(* Call ST03_572_Y70_0  Zuführung Vereinzler AST/GST  (Valve) *)
Analyze(InputExp:=  TRUE, DoAnalyze:= TRUE );
ST03_572_Y70_0.strAnlayse:=Analyze.OutString;
ST03_572_Y70_0(Enable  :=  Analyze.ExpResult,
                                sVisu:=Visu.ST03_572_Y70_0,
                                Reset:=gResetAll,
);
ST03_571_B69_2(ValveObject:= ADR(ST03_572_Y70_0));(*  Zuführung Vereinzler eingefahren GST*)
ST03_571_B69_3(ValveObject:= ADR(ST03_572_Y70_0));(*  Zuführung Vereinzler ausgefahren AST*)

(* Call ST03_572_Y70_1  Züführung Stopper AST/GST  (Valve) *)
Analyze(InputExp:=  TRUE, DoAnalyze:= TRUE );
ST03_572_Y70_1.strAnlayse:=Analyze.OutString;
ST03_572_Y70_1(Enable  :=  Analyze.ExpResult,
                                sVisu:=Visu.ST03_572_Y70_1,
                                Reset:=gResetAll,
);
ST03_571_B69_4(ValveObject:= ADR(ST03_572_Y70_1));(* Zuführung Stopper  eingefahren  AST*)
ST03_571_B69_5(ValveObject:= ADR(ST03_572_Y70_1));(* Zuführung Stopper  ausgefahren GST*)


(* Call ST03_571_B69_6 SK anwesend am Stoper (DigIn) *)
ST03_571_B69_6(sVisu:=Visu.ST03_571_B69_6,
                                Reset:=gResetAll,
);
(* Call ST03_571_B69_7 ISK anwesend an Abholposition (DigIn) *)
ST03_571_B69_7(sVisu:=Visu.ST03_571_B69_7,
                                Reset:=gResetAll,
);
END_ACTION
ACTION call_46pol:
(* Call ST03_463_Y71_3 Förderband  Zuführung Vereinzler AST/GST  (Valve) *)
Analyze(InputExp:=  TRUE, DoAnalyze:= TRUE );
ST03_464_Y71_3.strAnlayse:=Analyze.OutString;
ST03_464_Y71_3(Enable  :=  Analyze.ExpResult,
                                sVisu:=Visu.ST03_464_Y71_3,
                                Reset:=gResetAll,
);
ST03_461_B69_0(ValveObject:= ADR(ST03_464_Y71_3));(*Förderband Zuführung Vereinzler   AST*)
ST03_461_B69_1(ValveObject:= ADR(ST03_464_Y71_3));(*Förderband Zuführung Vereinzler   GST*)

(* Call ST03_463_Y71_4 Förderband  Zuführung Stopper AST/GST  (Valve) *)
Analyze(InputExp:=  TRUE, DoAnalyze:= TRUE );
ST03_464_Y71_4.strAnlayse:=Analyze.OutString;
ST03_464_Y71_4(Enable  :=  Analyze.ExpResult,
                                sVisu:=Visu.ST03_464_Y71_4,
                                Reset:=gResetAll,
);
ST03_461_B69_2(ValveObject:= ADR(ST03_464_Y71_4));(*Förderband Zuführung Stopper   AST*)
ST03_461_B69_3(ValveObject:= ADR(ST03_464_Y71_4));(*Förderband Zuführung Stopper   GST*)

(* Call ST03_461_B69_4 Zuführung  frei zum Ablegen ISK SP Maschine Pos.1  (DigIn) *)
ST03_461_B69_4(sVisu:=Visu.ST03_461_B69_4,
                                Reset:=gResetAll,
);
(* Call ST03_461_B69_7 Zuführung  ISK anwesend am Stopper (DigIn) *)
ST03_461_B69_7(sVisu:=Visu.ST03_461_B69_7,
                                Reset:=gResetAll,
);
(* Call ST03_463_B70_7  ISK auf Übergabeposition zu Roboter  (DigIn) *)
ST03_463_B70_7(sVisu:=Visu.ST03_463_B70_7,
                                Reset:=gResetAll,
);
(* Call ST03_462_B70_0 Förderband  ISK anwesend Wender (DigIn) *)
ST03_462_B70_0(sVisu:=Visu.ST03_462_B70_0,
                                Reset:=gResetAll,
);
(* Call ST03_462_B70_1 Zuführung  ISK Lageerkennung rechts (DigIn) *)
ST03_462_B70_1(sVisu:=Visu.ST03_462_B70_1,
                                Reset:=gResetAll,
);
(* Call ST03_462_B70_2 Zuführung  ISK Lageerkennung links (DigIn) *)
ST03_462_B70_2(sVisu:=Visu.ST03_462_B70_2,
                                Reset:=gResetAll,
);
(* Call ST03_464_Y71_0 Förderband  Zuführung Vereinzelner Wender AST/GST  (Valve) *)
Analyze(InputExp:=  TRUE, DoAnalyze:= TRUE );
ST03_464_Y71_0.strAnlayse:=Analyze.OutString;
ST03_464_Y71_0(Enable  :=  Analyze.ExpResult,
                                sVisu:=Visu.ST03_464_Y71_0,
                                Reset:=gResetAll,
);
ST03_461_B69_5(ValveObject:= ADR(ST03_464_Y71_0));(*Förderbandeinheit  Zuführung  Vereinzelner Wender AST*)
ST03_461_B69_6(ValveObject:= ADR(ST03_464_Y71_0));(*Förderbandeinheit  Zuführung  Vereinzelner Wender GST*)

(* Call ST03_464_Y71_1 Förderband  Zuführung Zylinder Vakuumdüsen AST/GST  (Valve) *)
Analyze(InputExp:=  TRUE, DoAnalyze:= TRUE );
ST03_464_Y71_1.strAnlayse:=Analyze.OutString;
ST03_464_Y71_1(Enable  :=  Analyze.ExpResult,
                                sVisu:=Visu.ST03_464_Y71_1,
                                Reset:=gResetAll,
);
ST03_463_B70_3(ValveObject:= ADR(ST03_464_Y71_1));(*Förderband Zuführung Zylinder Vakuumdüsen   AST*)
ST03_463_B70_4(ValveObject:= ADR(ST03_464_Y71_1));(*Förderband Zuführung Zylinder Vakuumdüsen   GST*)

IF	ST03_463_B70_3.ValveSensor THEN
	ST03_463_B70_3_4_pos:= -14;
ELSIF
	ST03_463_B70_4.ValveSensor THEN
	ST03_463_B70_3_4_pos:= 0;
ELSE
	ST03_463_B70_3_4_pos:= -7;
END_IF

(* Call ST03_464_Y71_2  Förderband  Zuführung Wendestation Einlauf / Auslauf   (Valve) *)
Analyze(InputExp:=  TRUE, DoAnalyze:= TRUE );
ST03_464_Y71_2.strAnlayse:=Analyze.OutString;
ST03_464_Y71_2(Enable  :=  Analyze.ExpResult,
                                sVisu:=Visu.ST03_464_Y71_2,
                                Reset:=gResetAll,
);
ST03_463_B70_5(ValveObject:= ADR(ST03_464_Y71_2));(*Förderband Zuführung Wendestation   AST*)
ST03_463_B70_6(ValveObject:= ADR(ST03_464_Y71_2));(*Förderband Zuführung Wendestation   GST*)

(* Call ST03_464_Y71_5  Förderband  Zuführung Vakuumdüsen EIN/AUS  (Valve) *)
Analyze(InputExp:=  TRUE, DoAnalyze:= TRUE );
ST03_464_Y71_5.strAnlayse:=Analyze.OutString;
ST03_464_Y71_5(Enable  :=  Analyze.ExpResult,
                                sVisu:=Visu.ST03_464_Y71_5,
                                Reset:=gResetAll,
);
(* Call ST03_464_B71_6  Vakuum vorhanden (DigIn) *)
ST03_464_B71_6(sVisu:=Visu.ST03_464_B71_6,
                                Reset:=gResetAll,
);
(* Call ST03_464_B71_7 Förderband  Staustrecke mitte voll (DigIn) *)
ST03_464_B71_7(sVisu:=Visu.ST03_464_B71_7,
                                Reset:=gResetAll,
);
END_ACTION
ACTION call_48pol:
(* Call ST03_551_B69_0 IZuführung  frei zum Ablegen ISK SP Maschine (DigIn) *)
ST03_551_B69_0(sVisu:=Visu.ST03_551_B69_0,
                                Reset:=gResetAll,
);
(* Call ST03_552_Y70_1  Zuführung Vereinzler AST/GST  (Valve) *)
Analyze(InputExp:=  TRUE, DoAnalyze:= TRUE );
ST03_552_Y70_1.strAnlayse:=Analyze.OutString;
ST03_552_Y70_1(Enable  :=  Analyze.ExpResult,
                                sVisu:=Visu.ST03_552_Y70_1,
                                Reset:=gResetAll,
);
ST03_551_B69_1(ValveObject:= ADR(ST03_552_Y70_1));(*  Zuführung Vereinzler eingefahren GST*)
ST03_551_B69_2(ValveObject:= ADR(ST03_552_Y70_1));(*  Zuführung Vereinzler ausgefahren AST*)

(* Call ST03_552_Y70_2  Züführung Stopper AST/GST  (Valve) *)
Analyze(InputExp:=  TRUE, DoAnalyze:= TRUE );
ST03_552_Y70_2.strAnlayse:=Analyze.OutString;
ST03_552_Y70_2(Enable  :=  Analyze.ExpResult,
                                sVisu:=Visu.ST03_552_Y70_2,
                                Reset:=gResetAll,
);
ST03_551_B69_3(ValveObject:= ADR(ST03_552_Y70_2));(* Zuführung Stopper  eingefahren  AST*)
ST03_551_B69_4(ValveObject:= ADR(ST03_552_Y70_2));(* Zuführung Stopper  ausgefahren GST*)


(* Call ST03_551_B69_6 SK anwesend am Stoper (DigIn) *)
ST03_551_B69_6(sVisu:=Visu.ST03_551_B69_6,
                                Reset:=gResetAll,
);
(* Call ST03_541_B69_7 ISK Lageerkennung links (DigIn) *)
ST03_551_B69_7(sVisu:=Visu.ST03_551_B69_7,
                                Reset:=gResetAll,
);
(* Call ST03_542_B70_0  ISK Lageerkennung rechts (DigIn) *)
ST03_552_B70_0(sVisu:=Visu.ST03_552_B70_0,
                                Reset:=gResetAll,
);
END_ACTION
ACTION call_72pol:
(* Call ST03_546_B69_0 IZuführung  frei zum Ablegen ISK SP Maschine (DigIn) *)
ST03_546_B69_0(sVisu:=Visu.ST03_546_B69_0,
                                Reset:=gResetAll,
);
(* Call ST03_547_Y70_1  Zuführung Vereinzler AST/GST  (Valve) *)
Analyze(InputExp:=  TRUE, DoAnalyze:= TRUE );
ST03_547_Y70_1.strAnlayse:=Analyze.OutString;
ST03_547_Y70_1(Enable  :=  Analyze.ExpResult,
                                sVisu:=Visu.ST03_547_Y70_1,
                                Reset:=gResetAll,
);
ST03_546_B69_1(ValveObject:= ADR(ST03_547_Y70_1));(*  Zuführung Vereinzler eingefahren GST*)
ST03_546_B69_2(ValveObject:= ADR(ST03_547_Y70_1));(*  Zuführung Vereinzler ausgefahren AST*)

(* Call ST03_547_Y70_2  Züführung Stopper AST/GST  (Valve) *)
Analyze(InputExp:=  TRUE, DoAnalyze:= TRUE );
ST03_547_Y70_2.strAnlayse:=Analyze.OutString;
ST03_547_Y70_2(Enable  :=  Analyze.ExpResult,
                                sVisu:=Visu.ST03_547_Y70_2,
                                Reset:=gResetAll,
);
ST03_546_B69_3(ValveObject:= ADR(ST03_547_Y70_2));(* Zuführung Stopper  eingefahren  AST*)
ST03_546_B69_4(ValveObject:= ADR(ST03_547_Y70_2));(* Zuführung Stopper  ausgefahren GST*)


(* Call ST03_546_B69_6 SK anwesend am Stoper (DigIn) *)
ST03_546_B69_6(sVisu:=Visu.ST03_546_B69_6,
                                Reset:=gResetAll,
);
(* Call ST03_546_B69_7 ISK anwesend an Abholposition (DigIn) *)
ST03_546_B69_7(sVisu:=Visu.ST03_546_B69_7,
                                Reset:=gResetAll,
);
(* Call ST03_547_B70_0  ISK Lageerkennung (DigIn) *)
ST03_547_B70_0(sVisu:=Visu.ST03_547_B70_0,
                                Reset:=gResetAll,
);
END_ACTION
ACTION call_74_91_35_168_160pol:
(* Call ST03_421_B63_4 Förderband frei zum Ablegen ISK SP Maschine Pos1  (DigIn) *)
ST03_421_B63_4(sVisu:=Visu.ST03_421_B63_4,
                                Reset:=gResetAll,
);
(* Call ST03_421_B63_5 Förderband frei zum Ablegen ISK SP Maschine Pos2  (DigIn) *)
ST03_421_B63_5(sVisu:=Visu.ST03_421_B63_5,
                                Reset:=gResetAll,
);
(* Call ST03_421_B63_6 Förderband frei zum Ablegen ISK SP Maschine Pos3  (DigIn) *)
ST03_421_B63_6(sVisu:=Visu.ST03_421_B63_6,
                                Reset:=gResetAll,
);
(* Call ST03_421_B63_7 ISK anwesend am Vereinzler  (DigIn) *)
ST03_421_B63_7(sVisu:=Visu.ST03_421_B63_7,
                                Reset:=gResetAll,
);
(* Call ST03_422_B64_0 Förderband Trigger Tintenstrahldrucker (Lichtschranke)  (DigIn) *)
ST03_422_B64_0(sVisu:=Visu.ST03_422_B64_0,
                                Reset:=gResetAll,
);
(* Call ST03_423_B66_0 Förderband Trigger Tintenstrahldrucker (Lichtschranke)  (DigIn) *)
ST03_423_B66_0(sVisu:=Visu.ST03_423_B66_0,
                                Reset:=gResetAll,
);
(* Call ST03_8_B76_1 Förderband Trigger Tintenstrahldrucker (Lichtschranke)  (DigIn) 3621 *)
ST03_8_B76_1(sVisu:=Visu.ST03_8_B76_1,
                                Reset:=gResetAll,
);
(* Call ST03_8_B76_2 Förderband Trigger Tintenstrahldrucker (Lichtschranke)  (DigIn) 3621 *)
ST03_8_B76_2(sVisu:=Visu.ST03_8_B76_2,
                                Reset:=gResetAll,
);
(* Call ST03_422_B64_3  Förderband ISK anwesend Stopper Kamera  (DigIn) *)
ST03_422_B64_3(sVisu:=Visu.ST03_422_B64_3,
                                Reset:=gResetAll,
);
(* Call ST03_422_B64_4 Zuführung ISK auf Übergabeposition Robo Palettierer  (DigIn) *)
ST03_422_B64_4(sVisu:=Visu.ST03_422_B64_4,
                                Reset:=gResetAll,
);
(* Call ST03_422_Y64_5  Förderband  Zuführung Vereinzler AST/GST (Valve) *)
Analyze(InputExp:=  TRUE, DoAnalyze:= TRUE );
ST03_422_Y64_5.strAnlayse:=Analyze.OutString;
ST03_422_Y64_5(Enable  :=  Analyze.ExpResult,
                                sVisu:=Visu.ST03_422_Y64_5,
                                Reset:=gResetAll,
);
ST03_421_B63_0(ValveObject:= ADR(ST03_422_Y64_5));(*Förderband Zuführung Vereinzler AST*)
ST03_421_B63_1(ValveObject:= ADR(ST03_422_Y64_5));(*Förderband Zuführung Vereinzler GST*)

(* Call ST03_422_Y64_6 Förderband rechte Zuführung Vereinzler AST/GST (Valve) *)
Analyze(InputExp:=  TRUE, DoAnalyze:= TRUE );
ST03_422_Y64_6.strAnlayse:=Analyze.OutString;
ST03_422_Y64_6(Enable  :=  Analyze.ExpResult,
                                sVisu:=Visu.ST03_422_Y64_6,
                                Reset:=gResetAll,
);
ST03_421_B63_2(ValveObject:= ADR(ST03_422_Y64_6));(*Förderband Zuführung Stopper AST*)
ST03_421_B63_3(ValveObject:= ADR(ST03_422_Y64_6));(*Förderband Zuführung Stopper GST*)

(* Call ST03_422_Y64_7 Förderband links/rechts Züführung Stopper 1 AST/GST (Valve) *)
Analyze(InputExp:=  TRUE, DoAnalyze:= TRUE );
ST03_422_Y64_7.strAnlayse:=Analyze.OutString;
ST03_422_Y64_7(Enable  :=  Analyze.ExpResult,
                                sVisu:=Visu.ST03_422_Y64_7,
                                Reset:=gResetAll,
);
ST03_422_B64_2(ValveObject:= ADR(ST03_422_Y64_7));(*Förderband Zuführung Stopper Kamera AST*)
ST03_422_B64_1(ValveObject:= ADR(ST03_422_Y64_7));(*Förderband Zuführung Stopper Kamera GST*)


(* Call ST03_423_Y65_6 Förderband links/rechts Züführung Stopper 2 AST/GST (Valve) *)
Analyze(InputExp:=  TRUE, DoAnalyze:= TRUE );
ST03_423_Y65_6.strAnlayse:=Analyze.OutString;
ST03_423_Y65_6(Enable  :=  Analyze.ExpResult,
                                sVisu:=Visu.ST03_423_Y65_6,
                                Reset:=gResetAll,
);
ST03_423_B65_1(ValveObject:= ADR(ST03_423_Y65_6));(*Förderband Zuführung Stopper Kamera AST*)
ST03_423_B65_0(ValveObject:= ADR(ST03_423_Y65_6));(*Förderband Zuführung Stopper Kamera GST*)

(* Call ST03_423_Y65_7 Förderband links/rechts Züführung Stopper 3 AST/GST (Valve) *)
Analyze(InputExp:=  TRUE, DoAnalyze:= TRUE );
ST03_423_Y65_7.strAnlayse:=Analyze.OutString;
ST03_423_Y65_7(Enable  :=  Analyze.ExpResult,
                                sVisu:=Visu.ST03_423_Y65_7,
                                Reset:=gResetAll,
);
ST03_423_B65_3(ValveObject:= ADR(ST03_423_Y65_7));(*Förderband Zuführung Stopper Kamera AST*)
ST03_423_B65_4(ValveObject:= ADR(ST03_423_Y65_7));(*Förderband Zuführung Stopper Kamera GST*)

(* Call ST03_33F4 Steckdosenleise Tintenstrahldrucker  (DigIn) *)
ST03_33F4(		sVisu:=Visu.ST03_33F4,
				Reset:=gResetAll,
);
(* Call ST03_70U3_1 Bereit/ Im Druck Tintenstrahldrucker Frontseite   (DigIn) *)
ST03_70U3_1(sVisu:=Visu.ST03_70U3_1,
                                Reset:=gResetAll,
);
(* Call ST03_70U3_2 Tank voll Tintenstrahldrucker Frontseite   (DigIn) *)
ST03_70U3_2(	sVisu:=Visu.ST03_70U3_2,
				Reset:=gResetAll,
);
(* Call ST03_70U3_3 Fehler/Störung Tintenstrahldrucker Frontseite   (DigIn) *)
ST03_70U3_3(	sVisu:=Visu.ST03_70U3_3,
				Reset:=gResetAll,
);
(* Call ST03_71U3_1 Bereit/ Im Druck Tintenstrahldrucker Rückseite   (DigIn) *)
ST03_71U3_1(sVisu:=Visu.ST03_71U3_1,
                                Reset:=gResetAll,
);
(* Call ST03_71U3_2 Tank voll Tintenstrahldrucker Rückseite   (DigIn) *)
ST03_71U3_2(	sVisu:=Visu.ST03_71U3_2,
				Reset:=gResetAll,
);
(* Call ST03_71U3_3 Fehler/Störung Tintenstrahldrucker Rückseite   (DigIn) *)
ST03_71U3_3(	sVisu:=Visu.ST03_71U3_3,
				Reset:=gResetAll,
);
(* Call ST03_PLAN_70V1_1 Start  Bedrucken Tintenstrahldrucker Frontseite (DigOutIn) *)
ST03_PLAN_70V1_1(	sVisu:=Visu.ST03_PLAN_70V1_1,
						Reset:=gResetAll,
);
(* Call ST03_PLAN_70V1_1 Start  Bedrucken Tintenstrahldrucker Rückseite (DigOutIn) *)
ST03_PLAN_71V1_2(	sVisu:=Visu.ST03_PLAN_71V1_2,
						Reset:=gResetAll,
);
IF NOT MP.ST02.SensopartEthernet THEN
	(**Sensopart Kamera links*)
	ST03_8_80_A1(
		b_kamera_aktiv:=MP.ST03.FrontCamOn,
		st_Description:= 'Sensopart Kamera links',
		b_reset:=gResetAll );

	(**Sensopart Kamera rechts*)
	ST03_8_85_A1(
		b_kamera_aktiv:=MP.ST03.BackCamOn,
		st_Description:= 'Sensopart Kamera rechts',
		b_reset:=gResetAll );
ELSE
	(**Sensopart Kamera links*)
	IF MP.ST02.SensopartIPAdress <>''  THEN
		ST03_8_90_A1(
				Activated := MP.ST03.FrontCamOn,
				st_Description:= 'Sensopart Kamera links',
				);
		ST03_8_90_A1.s_IpAdress := MP.ST02.SensopartIPAdress;
		ST03_8_90_A1.i_CmdPort := 2006;
		ST03_8_90_A1.i_DataPort :=2005;
END_IF
	(**Sensopart Kamera rechts*)
	IF MP.ST02.SensopartIPAdress2 <>''  THEN
		ST03_8_95_A1(
				Activated := MP.ST03.BackCamOn,
				st_Description:= 'Sensopart Kamera rechts',
				);
		ST03_8_95_A1.s_IpAdress := MP.ST02.SensopartIPAdress2;
		ST03_8_95_A1.i_CmdPort := 2006;
		ST03_8_95_A1.i_DataPort :=2005;
	END_IF
END_IF

(* Init ST03_S18 ST02 Druckschalter Wartungseinheit Hauptluft Tintenstrahldrucker min.6 bar (DigIn)
nur bei 160 pol*)	
ST03_S18(	sVisu:=Visu.ST03_S18,
			Reset:=gResetAll,
);
(* Call ST03_H6 Signalsäule GR Bedruckung IO(DigOutIn) *)
ST03_H6(	sVisu:=Visu.ST03_H6,
			Reset:=gResetAll,
);
(* Call ST03_H7 Signalsäule RD Sammelstörung Bedruckung IO(DigOutIn) *)
ST03_H7(	sVisu:=Visu.ST03_H7,
			Reset:=gResetAll,
);
END_ACTION
ACTION call_7pol:
(* Call ST03_512_XG1 Zuführung  frei zum Ablegen ISK SP Maschine (DigIn) *)
ST03_512_XG1(sVisu:=Visu.ST03_512_XG1,
                                Reset:=gResetAll,
);
(* Call ST03_515_Y72_0 ISK Klemmer 1 AST/GST  (Valve) *)
Analyze(InputExp:=  TRUE, DoAnalyze:= TRUE );
ST03_515_Y72_0.strAnlayse:=Analyze.OutString;
ST03_515_Y72_0(Enable  :=  Analyze.ExpResult,
                                sVisu:=Visu.ST03_515_Y72_0,
                                Reset:=gResetAll,
);
ST03_512_B69_1(ValveObject:= ADR(ST03_515_Y72_0));(*ISK Klemmer 2 GST*)
ST03_512_B69_2(ValveObject:= ADR(ST03_515_Y72_0));(*ISK Klemmer 2 AST*)
ST03_512_B69_3(ValveObject:= ADR(ST03_515_Y72_0));(*ISK Klemmer 1 GST*)
ST03_512_B69_4(ValveObject:= ADR(ST03_515_Y72_0));(*ISK Klemmer 1 AST*)

(* Call ST03_515_Y72_1 Rinne schwenkern AST/GST  (Valve) *)
Analyze(InputExp:=  TRUE, DoAnalyze:= TRUE );
ST03_515_Y72_1.strAnlayse:=Analyze.OutString;
ST03_515_Y72_1(Enable  :=  Analyze.ExpResult,
                                sVisu:=Visu.ST03_515_Y72_1,
                                Reset:=gResetAll,
);
ST03_512_B69_5(ValveObject:= ADR(ST03_515_Y72_1));(*ISK Klemmer schwenkern 0° AST*)
ST03_512_B69_6(ValveObject:= ADR(ST03_515_Y72_1));(*ISK Klemmer schwenkern 180° GST*)

(* Call ST03_514_B71_7 Führungsschiene frei zum schwenken (DigIn) *)
ST03_514_B71_7(sVisu:=Visu.ST03_514_B71_7,
                                Reset:=gResetAll,
);
(* Call ST03_515_Y72_2 Führungsschiene  Zuführung Vereinzler AST/GST  (Valve) *)
Analyze(InputExp:=  TRUE, DoAnalyze:= TRUE );
ST03_515_Y72_2.strAnlayse:=Analyze.OutString;
ST03_515_Y72_2(Enable  :=  Analyze.ExpResult,
                                sVisu:=Visu.ST03_515_Y72_2,
                                Reset:=gResetAll,
);
ST03_513_B70_0(ValveObject:= ADR(ST03_515_Y72_2));(*Führungsschiene  Zuführung Vereinzler AST*)
ST03_513_B70_1(ValveObject:= ADR(ST03_515_Y72_2));(*Führungsschiene  Zuführung Vereinzler GST*)

(* Call ST03_515_Y72_3 Führungsschiene  Zuführung Stopper AST/GST  (Valve) *)
Analyze(InputExp:=  TRUE, DoAnalyze:= TRUE );
ST03_515_Y72_3.strAnlayse:=Analyze.OutString;
ST03_515_Y72_3(Enable  :=  Analyze.ExpResult,
                                sVisu:=Visu.ST03_515_Y72_3,
                                Reset:=gResetAll,
);
ST03_513_B70_2(ValveObject:= ADR(ST03_515_Y72_3));(*Führungsschiene  Zuführung Stopper AST*)
ST03_513_B70_3(ValveObject:= ADR(ST03_515_Y72_3));(*Führungsschiene  Zuführung Stopper GST*)

(* Call ST03_513_B70_4 ISK anwesend am Stopper(DigIn) *)
ST03_513_B70_4(sVisu:=Visu.ST03_513_B70_4,
                                Reset:=gResetAll,
);
(* Call ST03_515_Y72_4 Übergabeposition Stopper 1 AST/GST  (Valve) *)
Analyze(InputExp:=  TRUE, DoAnalyze:= TRUE );
ST03_515_Y72_4.strAnlayse:=Analyze.OutString;
ST03_515_Y72_4(Enable  :=  Analyze.ExpResult,
                                sVisu:=Visu.ST03_515_Y72_4,
                                Reset:=gResetAll,
);
ST03_513_B70_5(ValveObject:= ADR(ST03_515_Y72_4));(*Übergabeposition Stopper 1 AST*)
ST03_513_B70_6(ValveObject:= ADR(ST03_515_Y72_4));(*Übergabeposition Stopper 1 GST*)

(* Call ST03_513_B70_7 ISK auf Übergabeposition 1 (DigIn) *)
ST03_513_B70_7(sVisu:=Visu.ST03_513_B70_7,
                                Reset:=gResetAll,
);
(* Call ST03_515_Y72_5 Übergabeposition Stopper 2 AST/GST  (Valve) *)
Analyze(InputExp:=  TRUE, DoAnalyze:= TRUE );
ST03_515_Y72_5.strAnlayse:=Analyze.OutString;
ST03_515_Y72_5(Enable  :=  Analyze.ExpResult,
                                sVisu:=Visu.ST03_515_Y72_5,
                                Reset:=gResetAll,
);
ST03_514_B71_0(ValveObject:= ADR(ST03_515_Y72_5));(*Übergabeposition Stopper 2 AST*)
ST03_514_B71_1(ValveObject:= ADR(ST03_515_Y72_5));(*Übergabeposition Stopper 2 GST*)

(* Call ST03_514_B71_2 ISK auf Übergabeposition 2 (DigIn) *)
ST03_514_B71_2(sVisu:=Visu.ST03_514_B71_2,
                                Reset:=gResetAll,
);
(* Call ST03_515_Y72_6 Übergabeposition Stopper 3 AST/GST  (Valve) *)
Analyze(InputExp:=  TRUE, DoAnalyze:= TRUE );
ST03_515_Y72_6.strAnlayse:=Analyze.OutString;
ST03_515_Y72_6(Enable  :=  Analyze.ExpResult,
                                sVisu:=Visu.ST03_515_Y72_6,
                                Reset:=gResetAll,
);
ST03_514_B71_3(ValveObject:= ADR(ST03_515_Y72_6));(*Übergabeposition Stopper 3 AST*)
ST03_514_B71_4(ValveObject:= ADR(ST03_515_Y72_6));(*Übergabeposition Stopper 3 GST*)

(* Call ST03_514_B71_5 ISK auf Übergabeposition 3 (DigIn) *)
ST03_514_B71_5(sVisu:=Visu.ST03_514_B71_5,
                                Reset:=gResetAll,
);
(* Call ST03_514_B71_6 ISK auf Übergabeposition 4 (DigIn) *)
ST03_514_B71_6(sVisu:=Visu.ST03_514_B71_6,
                                Reset:=gResetAll,
);
END_ACTION
ACTION call_88pol:
(* Call ST03_501_B69_0 IZuführung  frei zum Ablegen ISK SP Maschine (DigIn) *)
ST03_501_B69_0(sVisu:=Visu.ST03_501_B69_0,
                                Reset:=gResetAll,
);
(* Call ST03_502_Y70_1 Förderband  Zuführung Vereinzler AST/GST  (Valve) *)
Analyze(InputExp:=  TRUE, DoAnalyze:= TRUE );
ST03_502_Y70_1.strAnlayse:=Analyze.OutString;
ST03_502_Y70_1(Enable  :=  Analyze.ExpResult,
                                sVisu:=Visu.ST03_502_Y70_1,
                                Reset:=gResetAll,
);
ST03_501_B69_1(ValveObject:= ADR(ST03_502_Y70_1));(*Förderband Zuführung Vereinzler   AST*)
ST03_501_B69_2(ValveObject:= ADR(ST03_502_Y70_1));(*Förderband Zuführung Vereinzler   GST*)

(* Call ST03_502_Y70_2 örderband  Züführung Stopper AST/GST  (Valve) *)
Analyze(InputExp:=  TRUE, DoAnalyze:= TRUE );
ST03_502_Y70_2.strAnlayse:=Analyze.OutString;
ST03_502_Y70_2(Enable  :=  Analyze.ExpResult,
                                sVisu:=Visu.ST03_502_Y70_2,
                                Reset:=gResetAll,
);
ST03_501_B69_3(ValveObject:= ADR(ST03_502_Y70_2));(*Förderband Zuführung Stopper   AST*)
ST03_501_B69_4(ValveObject:= ADR(ST03_502_Y70_2));(*Förderband Zuführung Stopper   GST*)

(* Call ST03_501_B69_5 SK anwesend am Vereinzler (DigIn) *)
ST03_501_B69_5(sVisu:=Visu.ST03_501_B69_5,
                                Reset:=gResetAll,
);
(* Call ST03_501_B69_6 SK anwesend am Stoper (DigIn) *)
ST03_501_B69_6(sVisu:=Visu.ST03_501_B69_6,
                                Reset:=gResetAll,
);
(* Call ST03_501_B69_7 ISK auf Abholposition Robi (DigIn) *)
ST03_501_B69_7(sVisu:=Visu.ST03_501_B69_7,
                                Reset:=gResetAll,
);
(* Call ST03_502_B70_0  ISK Lageerkennung (DigIn) *)
ST03_502_B70_0(sVisu:=Visu.ST03_502_B70_0,
                                Reset:=gResetAll,
);
END_ACTION
ACTION call_88polAMG:
(* Call ST03_521_B69_0 IZuführung  frei zum Ablegen ISK SP Maschine (DigIn) *)
ST03_521_B69_0(sVisu:=Visu.ST03_521_B69_0,
                                Reset:=gResetAll,
);
(* Call ST03_522_Y70_1  Zuführung Vereinzler AST/GST  (Valve) *)
Analyze(InputExp:=  TRUE, DoAnalyze:= TRUE );
ST03_522_Y70_1.strAnlayse:=Analyze.OutString;
ST03_522_Y70_1(Enable  :=  Analyze.ExpResult,
                                sVisu:=Visu.ST03_522_Y70_1,
                                Reset:=gResetAll,
);
ST03_521_B69_1(ValveObject:= ADR(ST03_522_Y70_1));(*  Zuführung Vereinzler eingefahren GST*)
ST03_521_B69_2(ValveObject:= ADR(ST03_522_Y70_1));(*  Zuführung Vereinzler ausgefahren AST*)

(* Call ST03_522_Y70_2  Züführung Stopper AST/GST  (Valve) *)
Analyze(InputExp:=  TRUE, DoAnalyze:= TRUE );
ST03_522_Y70_2.strAnlayse:=Analyze.OutString;
ST03_522_Y70_2(Enable  :=  Analyze.ExpResult,
                                sVisu:=Visu.ST03_522_Y70_2,
                                Reset:=gResetAll,
);
ST03_521_B69_3(ValveObject:= ADR(ST03_522_Y70_2));(* Zuführung Stopper  eingefahren  AST*)
ST03_521_B69_4(ValveObject:= ADR(ST03_522_Y70_2));(* Zuführung Stopper  ausgefahren GST*)


(* Call ST03_521_B69_6 SK anwesend am Stoper (DigIn) *)
ST03_521_B69_6(sVisu:=Visu.ST03_521_B69_6,
                                Reset:=gResetAll,
);
(* Call ST03_521_B69_7 ISK Lageerkennung links (DigIn) *)
ST03_521_B69_7(sVisu:=Visu.ST03_521_B69_7,
                                Reset:=gResetAll,
);
(* Call ST03_522_B70_0  ISK Lageerkennung rechts (DigIn) *)
ST03_522_B70_0(sVisu:=Visu.ST03_522_B70_0,
                                Reset:=gResetAll,
);
END_ACTION
ACTION call_92pol:
(* Call ST03_446_Y70_5 Förderband  Zuführung Vereinzler AST/GST  (Valve) *)
Analyze(InputExp:=  TRUE, DoAnalyze:= TRUE );
ST03_446_Y70_5.strAnlayse:=Analyze.OutString;
ST03_446_Y70_5(Enable  :=  Analyze.ExpResult,
                                sVisu:=Visu.ST03_446_Y70_5,
                                Reset:=gResetAll,
);
ST03_444_B69_0(ValveObject:= ADR(ST03_446_Y70_5));(*Förderband Zuführung Vereinzler   AST*)
ST03_444_B69_1(ValveObject:= ADR(ST03_446_Y70_5));(*Förderband Zuführung Vereinzler   GST*)

(* Call ST03_446_Y70_6 Förderband  Zuführung Stopper AST/GST  (Valve) *)
Analyze(InputExp:=  TRUE, DoAnalyze:= TRUE );
ST03_446_Y70_6.strAnlayse:=Analyze.OutString;
ST03_446_Y70_6(Enable  :=  Analyze.ExpResult,
                                sVisu:=Visu.ST03_446_Y70_6,
                                Reset:=gResetAll,
);
ST03_444_B69_2(ValveObject:= ADR(ST03_446_Y70_6));(*Förderband Zuführung Stopper   AST*)
ST03_444_B69_3(ValveObject:= ADR(ST03_446_Y70_6));(*Förderband Zuführung Stopper   GST*)

(* Call ST03_444_B69_4 Zuführung  frei zum Ablegen ISK SP Maschine Pos.1  (DigIn) *)
ST03_444_B69_4(sVisu:=Visu.ST03_444_B69_4,
                                Reset:=gResetAll,
);
(* Call ST03_444_B69_7 Zuführung  ISK anwesend am Stopper (DigIn) *)
ST03_444_B69_7(sVisu:=Visu.ST03_444_B69_7,
                                Reset:=gResetAll,
);
(* Call ST03_446_B70_4  ISK auf Übergabeposition zu Roboter  (DigIn) *)
ST03_446_B70_4(sVisu:=Visu.ST03_446_B70_4,
                                Reset:=gResetAll,
);
(* Call ST03_445_B70_1 Zuführung  ISK Lageerkennung links (DigIn) *)
ST03_445_B70_1(sVisu:=Visu.ST03_445_B70_1,
                                Reset:=gResetAll,
);
(* Call ST03_445_B70_2 Zuführung  ISK Lageerkennung links (DigIn) *)
ST03_445_B70_2(sVisu:=Visu.ST03_445_B70_2,
                                Reset:=gResetAll,
);
END_ACTION
ACTION call_NOX4pol:
ST03_8_100_A1(
		st_ctrl_in := ST03_8_100_A1.st_ctrl_in,
		Activated := MP.ST03.CamOn[1],
		st_Description:= 'Kamera Farberkennung',
		SensopartErgebnis:=TD.SensopartErgebnis,
		);
ST03_8_100_A1.s_IpAdress := MP.ST03.SensopartIPAdress[1];  		(* 'MP.SensopartIPAdress';*)
ST03_8_100_A1.i_CmdPort := 2006;
ST03_8_100_A1.i_DataPort :=2005;

(* Call ST03_492_Y70_0 Förderband  Zuführung Vereinzler AST/GST  (Valve) *)
Analyze(InputExp:=  TRUE, DoAnalyze:= TRUE );
ST03_492_Y70_0.strAnlayse:=Analyze.OutString;
ST03_492_Y70_0(Enable  :=  Analyze.ExpResult,
                                sVisu:=Visu.ST03_492_Y70_0,
                                Reset:=gResetAll,
);
ST03_491_B69_1(ValveObject:= ADR(ST03_492_Y70_0));(*Förderband Zuführung Vereinzler   AST*)
ST03_491_B69_2(ValveObject:= ADR(ST03_492_Y70_0));(*Förderband Zuführung Vereinzler   GST*)

(* Call ST03_492_Y70_1 Förderband  Zuführung Stopper AST/GST  (Valve) *)
Analyze(InputExp:=  TRUE, DoAnalyze:= TRUE );
ST03_492_Y70_1.strAnlayse:=Analyze.OutString;
ST03_492_Y70_1(Enable  :=  Analyze.ExpResult,
                                sVisu:=Visu.ST03_492_Y70_1,
                                Reset:=gResetAll,
);
ST03_491_B69_3(ValveObject:= ADR(ST03_492_Y70_1));(*Förderband Zuführung Stopper   AST*)
ST03_491_B69_4(ValveObject:= ADR(ST03_492_Y70_1));(*Förderband Zuführung Stopper   GST*)

(* Call ST03_491_B69_0 Zuführung  frei zum Ablegen ISK SP Maschine (DigIn) *)
ST03_491_B69_0(sVisu:=Visu.ST03_491_B69_0,
                                Reset:=gResetAll,
);
(* Call ST03_491_B69_5 SK anwesend am Stoper (DigIn) *)
ST03_491_B69_5(sVisu:=Visu.ST03_491_B69_5,
                                Reset:=gResetAll,
);
(* Call ST03_491_B69_7 ISK auf Abholposition Robi (DigIn) *)
ST03_491_B69_7(sVisu:=Visu.ST03_491_B69_7,
                                Reset:=gResetAll,
);
END_ACTION
ACTION call_NOX5_6pol:
(* Sensopart Kamera*)
ST03_8_100_A1(
		st_ctrl_in := ST03_8_100_A1.st_ctrl_in,
		st_Description:= 'Sensopart Kamera',
		st_InstName := 'ST03_8_100_A1',
		Activated := MP.ST03.CamOn[1],
		SensopartErgebnis:=TD.SensopartErgebnis,
		);
ST03_8_100_A1.s_IpAdress := MP.ST03.SensopartIPAdress[1];  		(* 'MP.SensopartIPAdress';*)
ST03_8_100_A1.i_CmdPort := 2006;
ST03_8_100_A1.i_DataPort :=2005;

(* Keyence Kamera*)
ST03_8_105_A1();

ST03_8_105_A1.sConfig.Description := 'Keyence Kamera';
ST03_8_105_A1.sConfig.InstName := 'ST03_8_105_A1';
ST03_8_105_A1.sConfig.Aktiv := MP.ST03.CamOn_KYE;


(* Call ST03_4x2_B69_0 Zuführung frei zum Ablegen ISK SP Maschine  (DigIn) *)
ST03_4x2_B69_0(sVisu:=Visu.ST03_4x2_B69_0,
                                Reset:=gResetAll,
);
(* Call ST03_4x2_B69_5 ISK anwesend am Stopper  (DigIn) *)
ST03_4x2_B69_5(sVisu:=Visu.ST03_4x2_B69_5,
                                Reset:=gResetAll,
);
(* Call ST03_4x3_B70_0 ISK anwesend Übergabeposition Stopper  (DigIn) *)
ST03_4x3_B70_0(sVisu:=Visu.ST03_4x3_B70_0,
                                Reset:=gResetAll,
);
(* Call ST03_4x3_B70_1 ISK anwesend Übergabeposition  (DigIn) *)
ST03_4x3_B70_1(sVisu:=Visu.ST03_4x3_B70_1,
                                Reset:=gResetAll,
);
(* Call ST03_4x3_Y70_5 Zuführung Vereinzler AST/GST  (Valve) *)
Analyze(InputExp:=  TRUE, DoAnalyze:= TRUE );
ST03_4x3_Y70_5.strAnlayse:=Analyze.OutString;
ST03_4x3_Y70_5(Enable  :=  Analyze.ExpResult,
                                sVisu:=Visu.ST03_4x3_Y70_5,
                                Reset:=gResetAll,
);
ST03_4x2_B69_1(ValveObject:= ADR(ST03_4x3_Y70_5));(*Zuführung Vereinzler GST eingefahren*)
ST03_4x2_B69_2(ValveObject:= ADR(ST03_4x3_Y70_5));(*Zuführung Vereinzler AST ausgefahren*)

(* Call ST03_4x3_Y70_6 Zuführung Stopper AST/GST  (Valve) *)
Analyze(InputExp:=  TRUE, DoAnalyze:= TRUE );
ST03_4x3_Y70_6.strAnlayse:=Analyze.OutString;
ST03_4x3_Y70_6(Enable  :=  Analyze.ExpResult,
                                sVisu:=Visu.ST03_4x3_Y70_6,
                                Reset:=gResetAll,
);
ST03_4x2_B69_3(ValveObject:= ADR(ST03_4x3_Y70_6));(*Zuführung Stopper AST eingefahren*)
ST03_4x2_B69_4(ValveObject:= ADR(ST03_4x3_Y70_6));(*Zuführung Stopper GST ausgefahren*)

(* Call ST03_4x3_Y70_7 Zuführung Stopper Übergabeposition AST/GST  (Valve) *)
Analyze(InputExp:=  TRUE, DoAnalyze:= TRUE );
ST03_4x3_Y70_7.strAnlayse:=Analyze.OutString;
ST03_4x3_Y70_7(Enable  :=  Analyze.ExpResult,
                                sVisu:=Visu.ST03_4x3_Y70_7,
                                Reset:=gResetAll,
);
ST03_4x2_B69_6(ValveObject:= ADR(ST03_4x3_Y70_7));(*Zuführung Stopper Übergabeposition AST eingefahren*)
ST03_4x2_B69_7(ValveObject:= ADR(ST03_4x3_Y70_7));(*Zuführung Stopper Übergabeposition GST ausgefahren*)
END_ACTION

(* POU Stations/ST_08_Palettierer/ST_08_CallFBs/ST08_CallFBs, ST *)
PROGRAM ST08_CallFBs


VAR


END_VAR
(*----------------------------------------------------------------------------------------------------------------------------------*)
(*Call ST08_180_M1 Abstapeln*)
ST08_180_M1.sConfig.Aktiv				:=MP.ST08.StapelMotor;
ST08_180_M1			(	sVisu:=Visu.ST08_180_M1,
						Override:= MP.ST08.Override_Abstapeln,
						Offset:=MP.ST08.PosOffsetAbstapeln.Pos,	(* in mm oder Grad am Antrieb*)
						Reset:=gResetAll,
						NotausOK := ST08_402_B51_4.BitInToCheck,
						sPosList:= TD.PosAbstapeln );
IF	ST08_180_M1.sVisuAxis.BtnTeach.Pressed THEN
	TD.PosAbstapeln[ST08_180_M1.sVisuAxis.PosNr].Pos:= STRING_TO_LREAL(LREAL_TO_FMTSTR(ST08_180_M1.sctrl.in.Position,2,TRUE));
END_IF
ST08_180_M1_ON	(
			b_Stop:= NOT ST08_402_B51_4.BitInToCheck ,
			Achse:=ST08_180_M1 );

(*Call ST08_185_M1 Aufstapeln*)
ST08_185_M1.sConfig.Aktiv				:=MP.ST08.StapelMotor;
ST08_185_M1			(	sVisu:=Visu.ST08_185_M1,
						Override:= MP.ST08.Override_Aufstapeln,
						Offset:=MP.ST08.PosOffsetAufstapeln.Pos,
						Reset:=gResetAll,
						NotausOK := ST08_402_B51_5.BitInToCheck,
						sPosList:= TD.PosAufstapeln);
IF	ST08_185_M1.sVisuAxis.BtnTeach.Pressed THEN
	TD.PosAufstapeln[ST08_185_M1.sVisuAxis.PosNr].Pos:= STRING_TO_LREAL(LREAL_TO_FMTSTR(ST08_185_M1.sctrl.in.Position,2,TRUE));
END_IF
ST08_185_M1_ON	(
			b_Stop:= NOT ST08_402_B51_5.BitInToCheck ,
			Achse:=ST08_185_M1 );

(*Call ST08_190_M1 Tray ausheben*)
ST08_190_M1.sConfig.Aktiv				:=MP.ST08.TrayAushebenMotor;
ST08_190_M1			(	sVisu:=Visu.ST08_190_M1,
						Override:= MP.ST08.Override_TrayAusheben,
						Offset:=MP.ST08.PosOffsetTrayAusheben.Pos,
						Reset:=gResetAll,
						NotausOK := ST00_350_B20_0.BitInToCheck,
						sPosList:= TD.PosTrayAusheben);
IF	ST08_190_M1.sVisuAxis.BtnTeach.Pressed THEN
	TD.PosAufstapeln[ST08_190_M1.sVisuAxis.PosNr].Pos:= STRING_TO_LREAL(LREAL_TO_FMTSTR(ST08_190_M1.sctrl.in.Position,2,TRUE));
END_IF
ST08_190_M1_ON	(
			b_Stop:= NOT ST00_350_B20_0.BitInToCheck ,
			Achse:=ST08_190_M1 );
(* ST08_190_M1 Tray ausheben --- Generating home position*)
IF MP.ST08.TrayAushebenMotor THEN
	gHomeOk:=gHomeOk AND ABS(ST08_190_M1.sPos.ist - TD.PosTrayAusheben[1].Pos) < 0.5; (*1=unten, 2=oben, *);
END_IF

(* Call ST08_400_B50_0 Traystapel vor Vereinzeler Einlaufband hinten (DigIn) *)
ST08_400_B50_0                 (sVisu:=Visu.ST08_400_B50_0,
                                Reset:=gResetAll,
);

(* Call ST08_401_B50_5 Traystapel vor Vereinzeler Einlaufband mitte (DigIn) *)
ST08_401_B50_5                 (sVisu:=Visu.ST08_401_B50_5,
                                Reset:=gResetAll,
);


(* Call ST08_402_B51_2  Traystapel vor Vereinzeler Einlaufband vorne (DigIn) *)
ST08_402_B51_2                 (sVisu:=Visu.ST08_402_B51_2,
                                Reset:=gResetAll,
);

(* Call ST08_402_B51_4 (* Luftzone 1 *) (DigIn) *)
ST08_402_B51_4                 (sVisu:=Visu.ST08_402_B51_4,
                                Reset:=gResetAll,
);
(* Call ST08_402_B51_5 (* Luftzone 2 *) (DigIn) *)
ST08_402_B51_5                 (sVisu:=Visu.ST08_402_B51_5,
                                Reset:=gResetAll,
);
(* Call ST08_404_B52_2 Traystapel in Ablageposition Isokörper (DigIn) *)
ST08_404_B52_2                 (sVisu:=Visu.ST08_404_B52_2,
                                Reset:=gResetAll,
);
(* Call ST08_404_B52_3 Traystapel richtig eingelegt Isokörper (DigIn) *)
ST08_404_B52_3                 (sVisu:=Visu.ST08_404_B52_3,
                                Reset:=gResetAll,
);

(* Call ST08_406_B54_3 Traystapel in Ausheber (DigIn) *)
ST08_406_B54_3                 (sVisu:=Visu.ST08_406_B54_3,
                                Reset:=gResetAll,
);
(* Call ST08_406_B54_0 Tray in Zwischenp. Entnahme Isokörper (Bandende) (DigIn) *)
ST08_406_B54_0                 (sVisu:=Visu.ST08_406_B54_0,
                                Reset:=gResetAll,
);

(* Call ST08_406_B54_6 Tray aus Entnahme ausgelaufen (Bandende) (DigIn) *)
ST08_406_B54_6                 (sVisu:=Visu.ST08_406_B54_6,
                                Reset:=gResetAll,
);

(* Call ST08_407_B55_4 Tray in Aufstapelposition eingelaufen STN8 (DigIn) *)
ST08_407_B55_4                 (sVisu:=Visu.ST08_407_B55_4,
                                Reset:=gResetAll,
);
(* Call ST08_409_B55_5 Auslaufrollenbahn voll STN8 (DigIn) *)
ST08_409_B55_5                 (sVisu:=Visu.ST08_409_B55_5,
                                Reset:=gResetAll,
);


(* Call ST08_412_B58_4 Rüstsatz Förderband frei zum Ablegen ISK von SP Maschine Position 1 (DigIn) *)
ST08_412_B58_4                 (sVisu:=Visu.ST08_412_B58_4,
                                Reset:=gResetAll,
);

(* Call ST08_412_B58_5 Rüstsatz Förderband frei zum Ablegen ISK von SP Maschine Position 2 (DigIn) *)
ST08_412_B58_5                 (sVisu:=Visu.ST08_412_B58_5,
                                Reset:=gResetAll,
);

(* Call ST08_412_B58_6 Rüstsatz Förderband frei zum Ablegen ISK von SP Maschine Position 3 (DigIn) *)
ST08_412_B58_6                 (sVisu:=Visu.ST08_412_B58_6,
                                Reset:=gResetAll,
);

(* Call ST08_412_B58_5_35pol Lageerkennung links (DigIn) *)
ST08_412_B58_5_35pol                 (sVisu:=Visu.ST08_412_B58_5_35pol,
                                Reset:=gResetAll,
);

(* Call ST08_412_B58_6_35pol Lageerkennung rechts (DigIn) *)
ST08_412_B58_6_35pol                 (sVisu:=Visu.ST08_412_B58_6_35pol,
                                Reset:=gResetAll,
);

(* Call ST08_412_B58_7 Rüstsatz Förderband  ISK anwesend zum Vereinzeln (DigIn) *)
ST08_412_B58_7                 (sVisu:=Visu.ST08_412_B58_7,
                                Reset:=gResetAll,
);

(* Call ST08_412_B59_0 Rüstsatz Förderband ISK auf Übergabeposition Roboter Verpackung (DigIn) *)
ST08_412_B59_0                 (sVisu:=Visu.ST08_412_B59_0,
                                Reset:=gResetAll,
);

(* Call ST08_169_K1 Bandantrieb 1 Auslauf leere Trays Ein (DigOutIn) *)
ST08_169_K1                    (sVisu:=Visu.ST08_169_K1,
                                Reset:=gResetAll,
);
(* Call ST08_169_K2 Bandantrieb 4 Auslauf leere Trays Ein (DigOutIn) *)
ST08_169_K2                    (sVisu:=Visu.ST08_169_K2,
                                Reset:=gResetAll,
);
(* Call ST08_170_K1 Bandantrieb 2 Hubquereinheit Trays Ein (DigOutIn) *)
ST08_170_K1                    (sVisu:=Visu.ST08_170_K1,
                                Reset:=gResetAll,
);
(* Call ST08_170_K2 Bandantrieb 3 Hubquereinheit Trays Ein (DigOutIn) *)
ST08_170_K2                    (sVisu:=Visu.ST08_170_K2,
                                Reset:=gResetAll,
);

IF MP.ST08.Trayzufuhr_Verlaengerung THEN
	(* Call ST08_400_Y50_0 Stopper Traystapel Einlaufb. hinten links + rechts AST (Valve) *)
	Analyze         (InputExp:=  TRUE,
	                 DoAnalyze:= TRUE );
	ST08_400_Y50_0.strAnlayse:=Analyze.OutString;
	ST08_400_Y50_0                 (Enable  :=  Analyze.ExpResult,
	                                sVisu:=Visu.ST08_400_Y50_0,
	                                Reset:=gResetAll,
	);
	ST08_400_B50_4(ValveObject:= ADR(ST08_400_Y50_0));(*ST08_400_B50_4 Stopper Traystapel Einlaufband hinten rechts GST*)
END_IF

(* Call ST08_400_Y50_2 Stopper Traystapel Einlaufb. mitte links + rechts AST (Valve) *)
Analyze         (InputExp:=  TRUE,
                 DoAnalyze:= TRUE );
ST08_400_Y50_2.strAnlayse:=Analyze.OutString;
ST08_400_Y50_2                 (Enable  :=  Analyze.ExpResult,
                                sVisu:=Visu.ST08_400_Y50_2,
                                Reset:=gResetAll,
);
ST08_401_B51_1(ValveObject:= ADR(ST08_400_Y50_2));(*ST08_400_B50_4 Stopper Traystapel Einlaufband mitte rechts GST*)

(* Call ST08_402_Y50_4 Stopper Traystapel Einlaufb. vorne links + rechts AST (Valve) *)
Analyze         (InputExp:=  TRUE,
                 DoAnalyze:= TRUE );
ST08_402_Y50_4.strAnlayse:=Analyze.OutString;
ST08_402_Y50_4                 (Enable  :=  Analyze.ExpResult,
                                sVisu:=Visu.ST08_402_Y50_4,
                                Reset:=gResetAll,
);
ST08_402_B51_6(ValveObject:= ADR(ST08_402_Y50_4));(*ST08_400_B50_4 Stopper Traystapel Einlaufband vorne rechts GST*)

(* Call ST08_403_Y50_6 Vakuum 1 Einlauf STN8 AST (Valve) *)
Analyze         (InputExp:=  TRUE,
                 DoAnalyze:= TRUE );
ST08_403_Y50_6.strAnlayse:=Analyze.OutString;
ST08_403_Y50_6                 (Enable  :=  Analyze.ExpResult,
                                sVisu:=Visu.ST08_403_Y50_6,
                                Reset:=gResetAll,
);

(* Call ST08_403_Y50_7 Vakuum 2 Einlauf STN8 AST (Valve) *)
Analyze         (InputExp:=  TRUE,
                 DoAnalyze:= TRUE );
ST08_403_Y50_7.strAnlayse:=Analyze.OutString;
ST08_403_Y50_7                 (Enable  :=  Analyze.ExpResult,
                                sVisu:=Visu.ST08_403_Y50_7,
                                Reset:=gResetAll,
);


(* Call ST08_405_Y51_0 Hubtüre 2 Einlauf Isokörper STN8 AST (Valve) *)
Analyze         (InputExp:=  TRUE,
                 DoAnalyze:= TRUE );
ST08_405_Y51_0.strAnlayse:=Analyze.OutString;
ST08_405_Y51_0                 (Enable  :=  Analyze.ExpResult,
                                sVisu:=Visu.ST08_405_Y51_0,
                                Reset:=gResetAll,
);

IF NOT MP.ST03.SGM_3621 THEN
	ST08_405_B53_6(ValveObject:= ADR(ST08_405_Y51_0));(*ST08_405_B53_6 Hubtüre 2 Einlauf STN8 AST*)
	ST08_405_B53_7(ValveObject:= ADR(ST08_405_Y51_0));(*ST08_405_B53_6 Hubtüre 2 Einlauf STN8 GST*)
ELSE
	ST08_405_B53_6(ValveObject:= ADR(ST08_405_Y51_0));(*ST08_405_B53_6 Hubtüre 2 Einlauf STN8 AST*)
END_IF

(* Call ST08_404_Y51_6 Stopper Traystapel Isokörper AST (Valve) *)
Analyze         (InputExp:=  TRUE,
                 DoAnalyze:= TRUE );
ST08_404_Y51_6.strAnlayse:=Analyze.OutString;
ST08_404_Y51_6                 (Enable  :=  Analyze.ExpResult,
                                sVisu:=Visu.ST08_404_Y51_6,
                                Reset:=gResetAll,
);
ST08_404_B52_4(ValveObject:= ADR(ST08_404_Y51_6));(*ST08_404_B52_4 Stopper Traystapel Isokörper AST*)
ST08_404_B52_5(ValveObject:= ADR(ST08_404_Y51_6));(*ST08_404_B52_5 Stopper Traystapel Isokörper GST*)

(* Call ST08_406_Y51_2 Hubtüre 3 STN8 AST (Valve) *)
Analyze         (InputExp:=  TRUE,
                 DoAnalyze:= TRUE );
ST08_406_Y51_2.strAnlayse:=Analyze.OutString;
ST08_406_Y51_2                 (Enable  :=  Analyze.ExpResult,
                                sVisu:=Visu.ST08_406_Y51_2,
                                Reset:=gResetAll,
);

IF NOT MP.ST03.SGM_3621 THEN
	ST08_407_B55_0(ValveObject:= ADR(ST08_406_Y51_2));(*ST08_407_B55_0 Hubtüre 3 Auslauf STN8 AST*)
	ST08_407_B55_1(ValveObject:= ADR(ST08_406_Y51_2));(*ST08_407_B55_0 Hubtüre 3 Auslauf STN8 GST*)
ELSE
	ST08_407_B55_0(ValveObject:= ADR(ST08_406_Y51_2));(*ST08_407_B55_0 Hubtüre 3 Auslauf STN8 AST*)
END_IF

(* Call ST08_407_Y51_4 Hubtüre 4 Auslauf STN8 AST (Valve) *)
Analyze         (InputExp:=  TRUE,
                 DoAnalyze:= TRUE );
ST08_407_Y51_4.strAnlayse:=Analyze.OutString;
ST08_407_Y51_4                 (Enable  :=  Analyze.ExpResult,
                                sVisu:=Visu.ST08_407_Y51_4,
                                Reset:=gResetAll,
);

IF NOT MP.ST03.SGM_3621 THEN
	ST08_407_B55_2(ValveObject:= ADR(ST08_407_Y51_4));(*ST08_407_B55_2 Hubtüre 4 Auslauf STN8 AST*)
	ST08_407_B55_3(ValveObject:= ADR(ST08_407_Y51_4));(*ST08_407_B55_2 Hubtüre 4 Auslauf STN8 GST*)
ELSE
	ST08_407_B55_2(ValveObject:= ADR(ST08_407_Y51_4));(*ST08_407_B55_2 Hubtüre 4 Auslauf STN8 AST*)
END_IF

(* Call ST08_406_Y52_3 Ausheber Trays Entnahmepos. Isok. STN8 GST (Valve) *)
Analyze         (InputExp:=  TRUE,
                 DoAnalyze:= TRUE );
ST08_406_Y52_3.strAnlayse:=Analyze.OutString;
ST08_406_Y52_3                 (Enable  :=  Analyze.ExpResult,
                                sVisu:=Visu.ST08_406_Y52_3,
                                Reset:=gResetAll,
);
ST08_406_B54_4(ValveObject:= ADR(ST08_406_Y52_3));(*ST08_406_B54_4 Ausheber Trays Entnahmepos. Isok. STN8 AST*)
ST08_406_B54_5(ValveObject:= ADR(ST08_406_Y52_3));(*ST08_406_B54_5 Ausheber Trays Entnahmepos. Isok. STN8 GST*)


IF NOT MP.ST03.SGM_3621 THEN
	(* Stopper links + rechts Traystapel Auslaufband einfahren (Valve) *)
	Analyze         (InputExp:=  TRUE,
	                 DoAnalyze:= TRUE );
	ST08_400_Y52_5.strAnlayse:=Analyze.OutString;
	ST08_400_Y52_5                 (Enable  :=  Analyze.ExpResult,
	                                sVisu:=Visu.ST08_400_Y52_5,
	                                Reset:=gResetAll,
	);

	ST08_400_B50_1(ValveObject:= ADR(ST08_400_Y52_5));(*ST08_400_B50_1 Stopper links + rechts Traystapel Auslaufband eingefahren*)
	ST08_400_B50_2(ValveObject:= ADR(ST08_400_Y52_5));(*ST08_400_B50_2 Stopper links + rechts Traystapel Auslaufband ausgefahren*)
	ST08_400_B50_3(ValveObject:= ADR(ST08_400_Y52_5));(*ST08_400_B50_3 Stopper links + rechts Traystapel Auslaufband eingefahren*)
	ST08_400_B50_6(ValveObject:= ADR(ST08_400_Y52_5));(*ST08_400_B50_6 Stopper links + rechts Traystapel Auslaufband ausgefahren*)
END_IF


IF MP.ST08.Traystapel_schieben THEN
	IF MP.ST08.Trayzufuhr_Verlaengerung THEN
		(* Call ST08_401_Y52_4 Traystapel schieben hinten ausfahren AST (Valve) *)
		Analyze         (InputExp:=  TRUE,
		                 DoAnalyze:= TRUE );
		ST08_401_Y52_4.strAnlayse:=Analyze.OutString;
		ST08_401_Y52_4                 (Enable  :=  Analyze.ExpResult,
		                                sVisu:=Visu.ST08_401_Y52_4,
		                                Reset:=gResetAll,
		);
		ST08_401_B50_7(ValveObject:= ADR(ST08_401_Y52_4));(*ST08_401_B50_7 Traystapel schieben hinten*)

		(* Call ST08_402_Y52_6 Traystapel schieben mitte ausfahren AST (Valve) *)
		Analyze         (InputExp:=  TRUE,
		                 DoAnalyze:= TRUE );
		ST08_402_Y52_6.strAnlayse:=Analyze.OutString;
		ST08_402_Y52_6                 (Enable  :=  Analyze.ExpResult,
		                                sVisu:=Visu.ST08_402_Y52_6,
		                                Reset:=gResetAll,
		);
		ST08_402_B51_3(ValveObject:= ADR(ST08_402_Y52_6));(*ST08_402_B51_3 Traystapel schieben mitte*)
	END_IF

	(* Call ST08_402_Y52_7 Traystapel schieben vorne ausfahren AST (Valve) *)
	Analyze         (InputExp:=  TRUE,
	                 DoAnalyze:= TRUE );
	ST08_402_Y52_7.strAnlayse:=Analyze.OutString;
	ST08_402_Y52_7                 (Enable  :=  Analyze.ExpResult,
	                                sVisu:=Visu.ST08_402_Y52_7,
	                                Reset:=gResetAll,
	);
	ST08_402_B51_7(ValveObject:= ADR(ST08_402_Y52_7));(*ST08_402_B51_7 Traystapel schieben vorne*)
END_IF


IF	NOT MP.ST08.StapelMotor THEN
	(* Call ST08_404_Y53_0 Abstapelzylinder 1 Isokörper AST (Valve) *)
	Analyze         (InputExp:=  TRUE,
	                 DoAnalyze:= TRUE );
	ST08_404_Y53_0.strAnlayse:=Analyze.OutString;
	ST08_404_Y53_0                 (Enable  :=  Analyze.ExpResult,
	                                sVisu:=Visu.ST08_404_Y53_0,
	                                Reset:=gResetAll,
	);
	ST08_404_B52_6(ValveObject:= ADR(ST08_404_Y53_0));(*ST08_404_B52_6 Abstapelzylinder 1 Isokörper AST*)
	ST08_404_B52_7(ValveObject:= ADR(ST08_404_Y53_0));(*ST08_404_B52_7 Abstapelzylinder 1 Isokörper GST*)

	
	(* Call ST08_404_Y53_2 Abstapelzylinder 2 Isokörper AST (Valve) *)
	Analyze         (InputExp:=  TRUE,
	                 DoAnalyze:= TRUE );
	ST08_404_Y53_2.strAnlayse:=Analyze.OutString;
	ST08_404_Y53_2                 (Enable  :=  Analyze.ExpResult,
	                                sVisu:=Visu.ST08_404_Y53_2,
	                                Reset:=gResetAll,
	);
	ST08_404_B53_0(ValveObject:= ADR(ST08_404_Y53_2));(*ST08_404_B53_0 Abstapelzylinder 2 Isokörper AST*)
	ST08_404_B53_1(ValveObject:= ADR(ST08_404_Y53_2));(*ST08_404_B53_1 Abstapelzylinder 2 Isokörper GST*)

	(* Call ST08_408_Y54_2 Abstapelzylinder 1 STN8 AST (Valve) *)
	Analyze         (InputExp:=  TRUE,
	                 DoAnalyze:= TRUE );
	ST08_408_Y54_2.strAnlayse:=Analyze.OutString;
	ST08_408_Y54_2                 (Enable  :=  Analyze.ExpResult,
	                                sVisu:=Visu.ST08_408_Y54_2,
	                                Reset:=gResetAll,
	);
	ST08_408_B56_4(ValveObject:= ADR(ST08_408_Y54_2));(*ST08_408_B56_4 Abstapelzylinder 1 STN8 AST*)
	ST08_408_B56_5(ValveObject:= ADR(ST08_408_Y54_2));(*ST08_408_B56_5 Abstapelzylinder 1 STN8 GST*)
	
	
	(* Call ST08_408_Y54_4 Abstapelzylinder 2 STN8 AST (Valve) *) 
	Analyze         (InputExp:=  TRUE,
	                 DoAnalyze:= TRUE );
	ST08_408_Y54_4.strAnlayse:=Analyze.OutString;
	ST08_408_Y54_4                 (Enable  :=  Analyze.ExpResult,
	                                sVisu:=Visu.ST08_408_Y54_4,
	                                Reset:=gResetAll,
	);
	ST08_408_B56_6(ValveObject:= ADR(ST08_408_Y54_4));(*ST08_408_B56_6 Abstapelzylinder 2 STN8 AST*)
	ST08_408_B56_7(ValveObject:= ADR(ST08_408_Y54_4));(*ST08_408_B56_7 Abstapelzylinder 2 STN8 GST*)
END_IF

(* Call ST08_405_Y53_4 Rückhaltezylinder li+re Traystapel Isokörper AST (Valve) *)
Analyze         (InputExp:=  TRUE,
                 DoAnalyze:= TRUE );
ST08_405_Y53_4.strAnlayse:=Analyze.OutString;
ST08_405_Y53_4                 (Enable  :=  Analyze.ExpResult,
                                sVisu:=Visu.ST08_405_Y53_4,
                                Reset:=gResetAll,
);
ST08_405_B53_2(ValveObject:= ADR(ST08_405_Y53_4));(*ST08_405_B53_2 Rückhaltezylinder links Traystapel Isokörper AST*)
ST08_405_B53_3(ValveObject:= ADR(ST08_405_Y53_4));(*ST08_405_B53_3 Rückhaltezylinder links Traystapel Isokörper GST*)
ST08_405_B53_4(ValveObject:= ADR(ST08_405_Y53_4));(*ST08_405_B53_4 Rückhaltezylinder links Traystapel Isokörper AST*)
ST08_405_B53_5(ValveObject:= ADR(ST08_405_Y53_4));(*ST08_405_B53_5 Rückhaltezylinder links Traystapel Isokörper GST*)



(* Call ST08_408_Y54_0 Rückhaltezylinder li.+re. Auslauf STN8 AST (Valve) *)
Analyze         (InputExp:=  TRUE,
                 DoAnalyze:= TRUE );
ST08_408_Y54_0.strAnlayse:=Analyze.OutString;
ST08_408_Y54_0                 (Enable  :=  Analyze.ExpResult,
                                sVisu:=Visu.ST08_408_Y54_0,
                                Reset:=gResetAll,
);
ST08_408_B56_0(ValveObject:= ADR(ST08_408_Y54_0));(*ST08_408_B56_0 Rückhaltezylinder links Traystapel Isokörper AST*)
ST08_408_B56_1(ValveObject:= ADR(ST08_408_Y54_0));(*ST08_408_B56_1 Rückhaltezylinder links Traystapel Isokörper GST*)
ST08_408_B56_2(ValveObject:= ADR(ST08_408_Y54_0));(*ST08_408_B56_2 Rückhaltezylinder links Traystapel Isokörper AST*)
ST08_408_B56_3(ValveObject:= ADR(ST08_408_Y54_0));(*ST08_408_B56_3 Rückhaltezylinder links Traystapel Isokörper GST*)


(* Call ST08_404_Y52_0 Hub Bandstrecke STN8 AST (Valve) *)
Analyze         (InputExp:=  TRUE,
                 DoAnalyze:= TRUE );
ST08_404_Y52_0.strAnlayse:=Analyze.OutString;
ST08_404_Y52_0                 (Enable  :=  Analyze.ExpResult,
                                sVisu:=Visu.ST08_404_Y52_0,
                                Reset:=gResetAll,
);
ST08_406_B54_1(ValveObject:= ADR(ST08_404_Y52_0));(*Hub Bandstrecke AST*)
ST08_406_B54_2(ValveObject:= ADR(ST08_404_Y52_0));(*Hub Bandstrecke AST*)

(* Rüstsatz Förderband Vereinzelner (Valve) *)
Analyze         (InputExp:=  TRUE,
                 DoAnalyze:= TRUE );
ST08_412_Y55_0.strAnlayse:=Analyze.OutString;
ST08_412_Y55_0                 (Enable  :=  Analyze.ExpResult,
                                sVisu:=Visu.ST08_412_Y55_0,
                                Reset:=gResetAll,
);

ST08_412_B58_0(ValveObject:= ADR(ST08_412_Y55_0));(*ST08_412_B58_0 Rüstsatz Förderband Vereinzelner eingefahren*)
ST08_412_B58_1(ValveObject:= ADR(ST08_412_Y55_0));(*ST08_412_B58_1 Rüstsatz Förderband Vereinzelner ausgefahren*)

(* Rüstsatz Förderband Stopper (Valve) *)
Analyze         (InputExp:=  TRUE,
                 DoAnalyze:= TRUE );
ST08_412_Y55_2.strAnlayse:=Analyze.OutString;
ST08_412_Y55_2                 (Enable  :=  Analyze.ExpResult,
                                sVisu:=Visu.ST08_412_Y55_2,
                                Reset:=gResetAll,
);

ST08_412_B58_2(ValveObject:= ADR(ST08_412_Y55_2));(*ST08_412_B58_2 Rüstsatz Förderband Stopper eingefahren*)
ST08_412_B58_3(ValveObject:= ADR(ST08_412_Y55_2));(*ST08_412_B58_3 Rüstsatz Förderband Stopper ausgefahren*)
END_PROGRAM

(* POU Stations/ST_00/ST00_SFCs/_CallSFCs, ST *)
PROGRAM _CallSFCs
VAR
	b_init							:BOOL:=FALSE;
	FBSocketCloseAll		:FB_SocketCloseAll;

END_VAR
IF	NOT b_init THEN
		FBSocketCloseAll(bExecute:=TRUE);
		IF	FBSocketCloseAll.bBusy THEN
			b_init:=TRUE;
		END_IF
ELSE
	FBSocketCloseAll(bExecute:=FALSE);
END_IF



ST00_CallSFCs();
ST02_CallSFCs();
ST03_CallSFCs();
ST08_CallSFCs();
END_PROGRAM

(* POU Stations/ST_00/ST00_SFCs/ST00_CallSFCs, ST *)
PROGRAM ST00_CallSFCs
VAR

END_VAR
CallSpecialModeSFCs();

HomePositionSFC();
(*ST00_LoadTInfo();*)
ST02_HomePosition();
ST03_HomePosition();
ST08_HomePosition();
END_PROGRAM

(* POU Stations/ST_02_RT_Tampondrucker/ST02_SFCs/ST02_CallSFCs, ST *)
PROGRAM ST02_CallSFCs

VAR
	fb_ton_wz	:TON;
END_VAR
fb_ton_wz(IN:= TRUE, PT:= t#30s , Q=> , ET=> );

(*Aufrufe nur wenn ein Tampondrucker angeschlossen ist, sonst kommen viele Fehlermeldungt*)
IF	gTypeCode=4991 OR		(*102pol*)
	gTypeCode=312	THEN	(*93pol*)
	ST02_Main();
	ST02_Main.FB_CurrentStepHistorie(st_CurrentStep:=ST02_Main.SFCCurrentStep);
	ST02_AutoStop();
	ST02_CallFBs();
END_IF
(*Sonst werden die Visuelemente nicht mit Texten befüllt*)
IF	ModeSelect.Mode<=MODE_MANUAL AND
	NOT fb_ton_wz.Q THEN
	ST02_CallFBs();
END_IF

	(*Sensopart Kamera initialisieren*)
IF 	NOT MP.ST02.SensopartEthernet THEN
	IF NOT ST02_DT_95_A1.b_ready THEN
		ST02_DT_95_A1.b_init := TRUE;
	ELSE
		ST02_DT_95_A1.b_init := FALSE;
	END_IF
ELSE
	(*Sensopart Kamera Ethernet initialisieren*)
	IF NOT ST02_DT_95_A2.st_ctrl_out.b_bereit AND MP.ST02.SensopartIPAdress <>''  THEN
		ST02_DT_95_A2.st_ctrl_in.b_init := TRUE;
	ELSE
		ST02_DT_95_A2.st_ctrl_in.b_init := FALSE;
	END_IF
END_IF
END_PROGRAM

(* POU Stations/ST_02_RT_Tampondrucker/ST02_FBs/ST02_CallFBs, ST *)
PROGRAM ST02_CallFBs
VAR

END_VAR
(*----------------------------------------------------------------------------------------------------------------------------------*)
(* ----------------------------------------------------------------------------------------- *)
(* Call ST02_FDB_40_B61 Iso von SPM auf Band abgelegt (DigIn) *)
ST02_FDB_40_B61                (sVisu:=Visu.ST02_FDB_40_B61,
                                Reset:=gResetAll,
			(*	CheckSignalHigh:=TRUE,*)
);
(* Call ST02_FDB_40_B71 ST02 Iso auf Band vor Vereinzler (DigIn) *)
ST02_FDB_40_B71                (sVisu:=Visu.ST02_FDB_40_B71,
                                Reset:=gResetAll,
			(*	CheckSignalHigh:=TRUE,*)
);
(* Call ST02_S1_6A01 ST02 Sicherung 24V (DigIn) *)
ST02_S1_6A01                (sVisu:=Visu.ST02_S1_6A01,
                                Reset:=gResetAll,
				CheckSignalHigh:=TRUE,
);

(*Sensopart Kamera für die Erkennung der Markierungen*)
ST02_DT_95_A1(
	b_kamera_aktiv:=MP.ST02.CamOn AND NOT MP.ST02.SensopartEthernet,
	st_Description:= 'Kamera Farberkennung',
	b_reset:=gResetAll );

(*Sensopart Kamera für die Erkennung der Markierungen*)
ST02_DT_95_A2(
	st_ctrl_in := ST02_DT_95_A2.st_ctrl_in,
	Activated := MP.ST02.CamOn AND MP.ST02.SensopartEthernet AND MP.ST02.SensopartIPAdress <> '',
	st_Description:= 'Kamera Farberkennung',
	);
IF 	MP.ST02.SensopartIPAdress <> ''  THEN
	ST02_DT_95_A2.s_IpAdress := MP.ST02.SensopartIPAdress;  		(* 'MP.SensopartIPAdress';*)
	ST02_DT_95_A2.i_CmdPort := 2006;
	ST02_DT_95_A2.i_DataPort :=2005;
END_IF

(* Call ST02_S1_70K61_A1 Start  Bedrucken (DigOutIn) *)
ST02_S1_70K61_A1                  (sVisu:=Visu.ST02_S1_70K61_A1,
                                Reset:=gResetAll,
);

(* Call ST02_62_Y6 Tisch drehen 0 - 180 Grad  (Valve) *)
Analyze         (InputExp:=  TRUE,
                 DoAnalyze:= TRUE );
ST02_62_Y6.strAnlayse:=Analyze.OutString;
ST02_62_Y6                 (Enable  :=  Analyze.ExpResult,
                                sVisu:=Visu.ST02_62_Y6,
                                Reset:=gResetAll,
);
ST02_DT_62_B81(ValveObject:= ADR(ST02_62_Y6));(*Tisch drehen 0 Grad*)
ST02_DT_62_B91(ValveObject:= ADR(ST02_62_Y6));(*Tisch drehen 180 Grad*)

IF	ST02_DT_62_B81.ValveSensor THEN
	MP.ST02.TableData[1].ProcessData.Nest_Nr:=2;
	MP.ST02.TableData[2].ProcessData.Nest_Nr:=1;
ELSIF	ST02_DT_62_B91.ValveSensor THEN
	MP.ST02.TableData[1].ProcessData.Nest_Nr:=1;
	MP.ST02.TableData[2].ProcessData.Nest_Nr:=2;
ELSE
	MP.ST02.TableData[1].ProcessData.Nest_Nr:=0;
	MP.ST02.TableData[2].ProcessData.Nest_Nr:=0;
END_IF
(*----------------------------------------------------------------------------------------------------------------------------------*)
(* Call ST02_62_Y9 Schwenkarm 2 drehen 90 - 180 Grad  (Valve) *)
Analyze         (InputExp:=  TRUE,
                 DoAnalyze:= TRUE );
ST02_62_Y9.strAnlayse:=Analyze.OutString;
ST02_62_Y9                 (Enable  :=  Analyze.ExpResult,
                                sVisu:=Visu.ST02_62_Y9,
                                Reset:=gResetAll,
);
(*ST02_DT_61_B21(ValveObject:= ADR(ST02_62_Y9));		(*Schwenkarm 2 90 Grad*)*)
ST02_DT_61_B11(ValveObject:= ADR(ST02_62_Y9));		(*Schwenkarm 2 180 Grad*)

(* Call ST02_62_Y11 Schwenkarm 2 drehen 90 - 0 Grad  (Valve) *)
Analyze         (InputExp:=  TRUE,
                 DoAnalyze:= TRUE );
ST02_62_Y11.strAnlayse:=Analyze.OutString;
ST02_62_Y11                 (Enable  :=  Analyze.ExpResult,
                                sVisu:=Visu.ST02_62_Y11,
                                Reset:=gResetAll,
);
(*ST02_DT_61_B21_clone(ValveObject:= ADR(ST02_62_Y11));(*Schwenkarm 2 90 Grad*)*)
ST02_DT_61_B31(ValveObject:= ADR(ST02_62_Y11));		(*Schwenkarm 2 0 Grad*)


ST02_Schwenkarm[2](
	ST02_90_180:=ST02_62_Y9 ,
	ST02_90_0:=ST02_62_Y11 ,
	ST02_90:=ST02_DT_61_B21);
(*----------------------------------------------------------------------------------------------------------------------------------*)
(* Call ST02_62_Y13 Schwenkarm 1 drehen 90 - 180 Grad  (Valve) *)
Analyze         (InputExp:=  TRUE,
                 DoAnalyze:= TRUE );
ST02_62_Y13.strAnlayse:=Analyze.OutString;
ST02_62_Y13                 (Enable  :=  Analyze.ExpResult,
                                sVisu:=Visu.ST02_62_Y13,
                                Reset:=gResetAll,
);
(*ST02_DT_61_B51(ValveObject:= ADR(ST02_62_Y13));		(*Schwenkarm 1 90 Grad*)*)
ST02_DT_61_B41(ValveObject:= ADR(ST02_62_Y13));		(*Schwenkarm 1 180 Grad*)

(* Call ST02_62_Y15 Schwenkarm 1 drehen 90 - 0 Grad  (Valve) *)
Analyze         (InputExp:=  TRUE,
                 DoAnalyze:= TRUE );
ST02_62_Y15.strAnlayse:=Analyze.OutString;
ST02_62_Y15                 (Enable  :=  Analyze.ExpResult,
                                sVisu:=Visu.ST02_62_Y15,
                                Reset:=gResetAll,
);
(*ST02_DT_61_B51_clone(ValveObject:= ADR(ST02_62_Y15));(*Schwenkarm 1 90 Grad*)*)
ST02_DT_62_B11(ValveObject:= ADR(ST02_62_Y15));		(*Schwenkarm 1 0 Grad*)

ST02_Schwenkarm[1](
	ST02_90_180:=ST02_62_Y13 ,
	ST02_90_0:=ST02_62_Y15,
	ST02_90:=ST02_DT_61_B51);

(* Call ST02_S1_40K01  Freigabe Förderband von SPM (DigIn) *)
ST02_S1_40K01                     (sVisu:=Visu.ST02_S1_40K01,
                                Reset:=gResetAll,
																CheckSignalHigh:=FALSE,
);
(* Call ST02_FDB_80_B02 Band Entnahmeposition 2 (DigIn) *)
ST02_FDB_80_B02                     (sVisu:=Visu.ST02_FDB_80_B02,
                                Reset:=gResetAll
);

(* Call ST02_FDB_54_B41 Kamera ISK anwesend an Prüfposition (DigIn) *)
ST02_FDB_54_B41               (sVisu:=Visu.ST02_FDB_54_B41,
                                Reset:=gResetAll,
);

(* Call ST02_DT_65B11 Tampondrucker Nest 1 leer (DigIn) *)
ST02_DT_65B11               (sVisu:=Visu.ST02_DT_65B11,
                                Reset:=gResetAll,
);

(* Call ST02_DT_65B21 Tampondrucker Nest 2 leer (DigIn) *)
ST02_DT_65B21               (sVisu:=Visu.ST02_DT_65B21,
                                Reset:=gResetAll,
);
(* Init ST02_35_S31 ST02 Druckschalter Wartungseinheit Hauptluft min.6 bar (DigIn) *)
ST02_35_S31 	                (sVisu:=Visu.ST02_35_S31,
                                Reset:=gResetAll,
			CheckSignalHigh:=TRUE,
);
(*----------------------------------------------------------------------------------------------------------------------------------*)
(* Call ST02_FDB_55X1_5_READY IFM Kamera Flügelerkennung links Ready (DigIn) *)
ST02_FDB_55X1_5_READY               (sVisu:=Visu.ST02_FDB_55X1_5_READY,
                                Reset:=gResetAll,
);
(* Call ST02_FDB_55X1_6_IO IFM Kamera Flügelerkennung links Ergebnis iO (DigIn) *)
ST02_FDB_55X1_6_IO               (sVisu:=Visu.ST02_FDB_55X1_6_IO,
                                Reset:=gResetAll,
);
(* Call ST02_FDB_55X1_6_NIO IFM Kamera Flügelerkennung links Ergebnis niO (DigIn) *)
ST02_FDB_55X1_6_NIO               (sVisu:=Visu.ST02_FDB_55X1_6_NIO,
                                Reset:=gResetAll,
);
(* Call ST02_FDB_55X1_2_TRIGGER IFM Kamera Flügelerkennung links Trigger (DigOutIn) *)
ST02_FDB_55X1_2_TRIGGER                  (sVisu:=Visu.ST02_FDB_55X1_2_TRIGGER,
                                Reset:=gResetAll,
);
(* Call ST02_FDB_55X1_7_JOB_BIT1 IFM Kamera  links Jobwechsel Bit1 (DigOutIn) *)
ST02_FDB_55X1_7_JOB_BIT1                  (sVisu:=Visu.ST02_FDB_55X1_7_JOB_BIT1,
                                Reset:=gResetAll,
);
(* Call ST02_FDB_55X1_7_JOB_BIT2 IFM Kamera  links Jobwechsel Bit2 (DigOutIn) *)
ST02_FDB_55X1_7_JOB_BIT2                  (sVisu:=Visu.ST02_FDB_55X1_7_JOB_BIT2,
                                Reset:=gResetAll,
);
(* Call ST02_FDB_56X1_5_READY IFM Kamera Flügelerkennung rechts Ready (DigIn) *)
ST02_FDB_56X1_5_READY               (sVisu:=Visu.ST02_FDB_56X1_5_READY,
                                Reset:=gResetAll,
);
(* Call ST02_FDB_56X1_6_IO IFM Kamera Flügelerkennung rechts Ergebnis iO (DigIn) *)
ST02_FDB_56X1_6_IO               (sVisu:=Visu.ST02_FDB_56X1_6_IO,
                                Reset:=gResetAll,
);
(* Call ST02_FDB_56X1_6_NIO IFM Kamera Flügelerkennung rechts Ergebnis niO (DigIn) *)
ST02_FDB_56X1_6_NIO               (sVisu:=Visu.ST02_FDB_56X1_6_NIO,
                                Reset:=gResetAll,
);
(* Call ST02_FDB_56X1_2_TRIGGER IFM Kamera Flügelerkennung rechts Trigger (DigOutIn) *)
ST02_FDB_56X1_2_TRIGGER                  (sVisu:=Visu.ST02_FDB_56X1_2_TRIGGER,
                                Reset:=gResetAll,
);
(* Call ST02_FDB_56X1_7_JOB_BIT1 IFM Kamera  rechts Jobwechsel Bit1 (DigOutIn) *)
ST02_FDB_56X1_7_JOB_BIT1                  (sVisu:=Visu.ST02_FDB_56X1_7_JOB_BIT1,
                                Reset:=gResetAll,
);
(* Call ST02_FDB_56X1_7_JOB_BIT2 IFM Kamera  rechts Jobwechsel Bit2 (DigOutIn) *)
ST02_FDB_56X1_7_JOB_BIT2                  (sVisu:=Visu.ST02_FDB_56X1_7_JOB_BIT2,
                                Reset:=gResetAll,
);
(* Call ST02_62_Y4 Kamera Ausschleusen Bandstrecke (Valve) *)
Analyze         (InputExp:=  TRUE,
                 DoAnalyze:= TRUE );
ST02_62_Y4.strAnlayse:=Analyze.OutString;
ST02_62_Y4                 (Enable  :=  Analyze.ExpResult,
                                sVisu:=Visu.ST02_62_Y4,
                                Reset:=gResetAll,
);
ST02_FDB_54_B11(ValveObject:= ADR(ST02_62_Y4));(*Kamera Ausschleusen Bandstrecke eingefahren*)
ST02_FDB_54_B21(ValveObject:= ADR(ST02_62_Y4));(*Kamera Ausschleusen Bandstrecke ausgefahren*)


(*Call ST02_62_Y17 Schwenkarm 1 ISK Fixierung ein/ausfahren(Valve) (Valve) *)
Analyze         (InputExp:=  TRUE,
                 DoAnalyze:= TRUE );
ST02_62_Y17.strAnlayse:=Analyze.OutString;
ST02_62_Y17                 (Enable  :=  Analyze.ExpResult,
                                sVisu:=Visu.ST02_62_Y17,
                                Reset:=gResetAll,
);
ST02_S1_66_B11(ValveObject:= ADR(ST02_62_Y17));(*Kamera Ausschleusen Bandstrecke eingefahren*)
ST02_S1_66_B21(ValveObject:= ADR(ST02_62_Y17));(*Kamera Ausschleusen Bandstrecke ausgefahren*)


(*Call ST02_62_Y18 Schwenkarm 2 ISK Fixierung ein/ausfahren(Valve) (Valve) *)
Analyze         (InputExp:=  TRUE,
                 DoAnalyze:= TRUE );
ST02_62_Y18.strAnlayse:=Analyze.OutString;
ST02_62_Y18                 (Enable  :=  Analyze.ExpResult,
                                sVisu:=Visu.ST02_62_Y18,
                                Reset:=gResetAll,
);
ST02_S1_66_B31(ValveObject:= ADR(ST02_62_Y18));(*Kamera Ausschleusen Bandstrecke eingefahren*)
ST02_S1_66_B41(ValveObject:= ADR(ST02_62_Y18));(*Kamera Ausschleusen Bandstrecke ausgefahren*)


(* Call ST02_35Y01 Einschaltventil Hauptluft Tampondruckanlage (Valve) *)
Analyze         (InputExp:=  TRUE,
                 DoAnalyze:= TRUE );
ST02_35Y01.strAnlayse:=Analyze.OutString;
ST02_35Y01               (Enable  :=  Analyze.ExpResult,
                                sVisu:=Visu.ST02_35Y01,
                                Reset:=gResetAll,
);
END_PROGRAM

(* POU Stations/ST_03_Ruestsaetze/ST_03_FBs/ST03_CallSFCs, ST *)
PROGRAM ST03_CallSFCs


VAR


END_VAR
ST03_Main();
ST03_Main.FB_CurrentStepHistorie(st_CurrentStep:=ST03_Main.SFCCurrentStep);


	(*Sensopart Kamera initialisieren*)
IF NOT MP.ST02.SensopartEthernet THEN
	IF NOT ST03_8_80_A1.b_ready THEN
		ST03_8_80_A1.b_init := TRUE;
	ELSE
		ST03_8_80_A1.b_init := FALSE;
	END_IF
	IF NOT ST03_8_85_A1.b_ready THEN
		ST03_8_85_A1.b_init := TRUE;
	ELSE
		ST03_8_85_A1.b_init := FALSE;
	END_IF
ELSE
	(*Sensopart Kamera Ethernet initialisieren*)
	IF NOT ST03_8_90_A1.st_ctrl_out.b_bereit AND MP.ST02.SensopartIPAdress <>''  THEN
		ST03_8_90_A1.st_ctrl_in.b_init := TRUE;
	ELSE
		ST03_8_90_A1.st_ctrl_in.b_init := FALSE;
	END_IF

	IF NOT ST03_8_95_A1.st_ctrl_out.b_bereit AND MP.ST02.SensopartIPAdress2 <>''  THEN
		ST03_8_95_A1.st_ctrl_in.b_init := TRUE;
	ELSE
		ST03_8_95_A1.st_ctrl_in.b_init := FALSE;
	END_IF

	IF NOT ST03_8_100_A1.st_ctrl_out.b_bereit AND MP.ST03.CamOn[1] THEN
		ST03_8_100_A1.st_ctrl_in.b_init := TRUE;
	ELSE
		ST03_8_100_A1.st_ctrl_in.b_init := FALSE;
	END_IF

	IF NOT ST03_8_103_A1.st_ctrl_out.b_bereit AND MP.ST03.CamOn[2] THEN
		ST03_8_103_A1.st_ctrl_in.b_init := TRUE;
	ELSE
		ST03_8_103_A1.st_ctrl_in.b_init := FALSE;
	END_IF

	(*Keyence Kamera Ethernet initialisieren*)
	IF NOT ST03_8_105_A1.st_ctrl_out.b_bereit AND MP.ST03.CamOn_KYE THEN
		ST03_8_105_A1.st_ctrl_in.b_init := TRUE;
	ELSE
		ST03_8_105_A1.st_ctrl_in.b_init := FALSE;
	END_IF


END_IF
END_PROGRAM

(* POU Stations/ST_08_Palettierer/ST_08_SFCs/ST08_CallSFCs, ST *)
 PROGRAM ST08_CallSFCs


VAR


END_VAR
ST08_Process();
ST08_Process.FB_CurrentStepHistorie(st_CurrentStep:=ST08_Process.SFCCurrentStep);

ST08_VV1_Y50_0();
ST08_VV1_Y50_2();

ST08_Depalletizing();
ST08_Depalletizing.FB_CurrentStepHistorie(st_CurrentStep:=ST08_Depalletizing.SFCCurrentStep);

ST08_Palletizing();
ST08_Palletizing.FB_CurrentStepHistorie(st_CurrentStep:=ST08_Palletizing.SFCCurrentStep);
END_PROGRAM

(* POU Stations/ST_08_Palettierer/ST_08_SFCs/Inlett/ST08_VV1_Y50_0, SFC *)
PROGRAM ST08_VV1_Y50_0				(* Vereinzler vor HQE4 *)

VAR_OUTPUT
	SFCCurrentPOU	: STRING:='ST08_VV1_Y50_0';
	SFCCurrentStep	: STRING:='';
	SFCTime			: DINT;
	State   		: DINT;
	Result  		: DINT;
END_VAR
VAR_INPUT

END_VAR
VAR
	MsgOK			: BOOL;
	MsgCancel		: BOOL;
	SFCRun			: BOOL;
	SFCTimeStart	: TIME;
	Delay			: TON;
	TimeOut			: TON;
	(* Userdefinded area *)

END_VAR
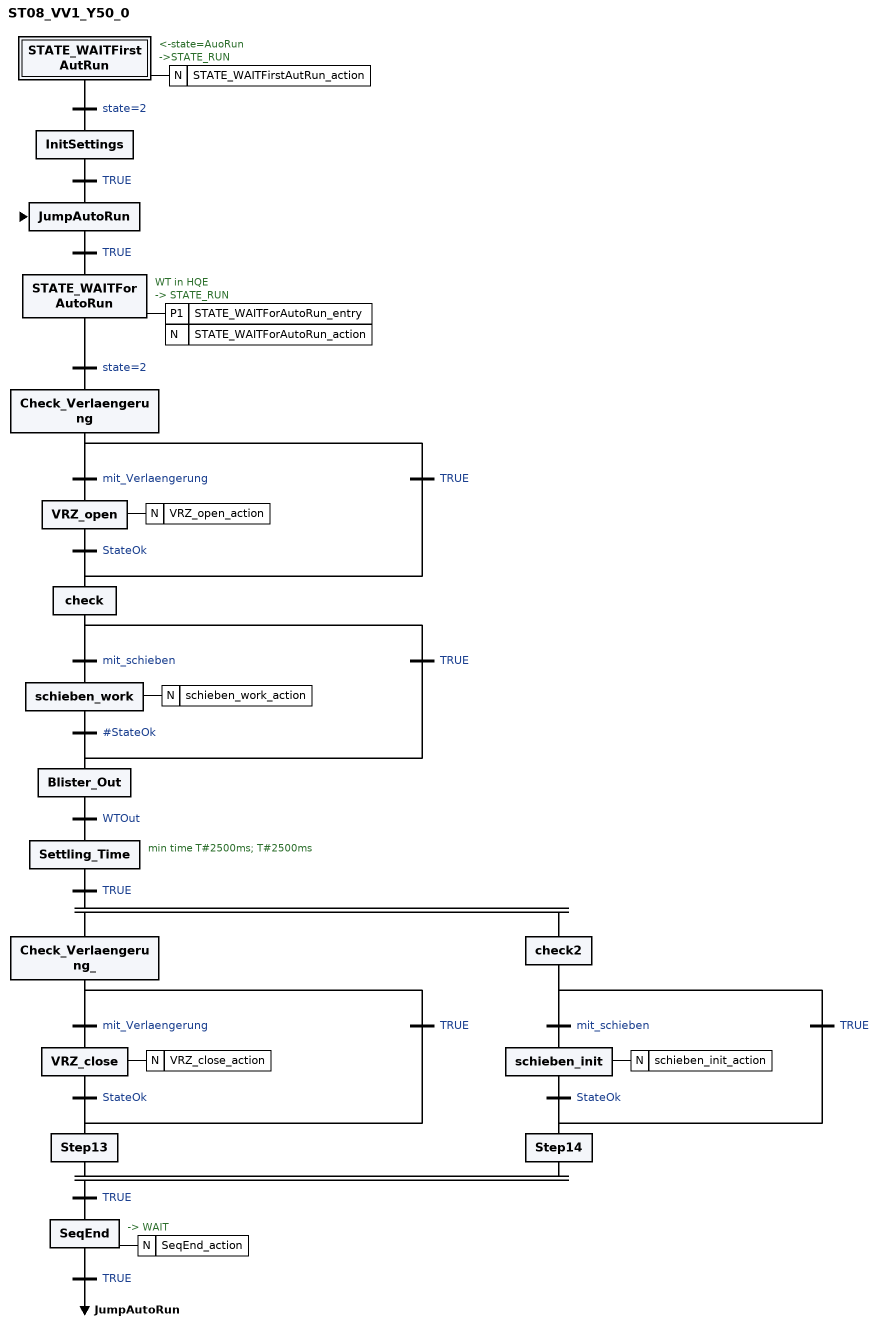
INITIAL_STEP STATE_WAITFirstAutRun: (* <-state=AuoRun / ->STATE_RUN *)
	STATE_WAITFirstAutRun_action(N);
END_STEP
TRANSITION FROM STATE_WAITFirstAutRun TO InitSettings := state=2;
END_TRANSITION
STEP InitSettings:
END_STEP
TRANSITION FROM InitSettings TO JumpAutoRun := TRUE;
END_TRANSITION
STEP JumpAutoRun:
END_STEP
TRANSITION FROM JumpAutoRun TO STATE_WAITForAutoRun := TRUE;
END_TRANSITION
STEP STATE_WAITForAutoRun: (* WT in HQE / -> STATE_RUN *)
	STATE_WAITForAutoRun_entry(P1);
	STATE_WAITForAutoRun_action(N);
END_STEP
TRANSITION FROM STATE_WAITForAutoRun TO Check_Verlaengerung := state=2;
END_TRANSITION
STEP Check_Verlaengerung:
END_STEP
TRANSITION FROM Check_Verlaengerung TO VRZ_open := mit_Verlaengerung;
END_TRANSITION
TRANSITION FROM Check_Verlaengerung TO check := TRUE;
END_TRANSITION
STEP VRZ_open:
	VRZ_open_action(N);
END_STEP
TRANSITION FROM VRZ_open TO check := StateOk;
END_TRANSITION
STEP check:
END_STEP
TRANSITION FROM check TO schieben_work := mit_schieben;
END_TRANSITION
TRANSITION FROM check TO Blister_Out := TRUE;
END_TRANSITION
STEP schieben_work:
	schieben_work_action(N);
END_STEP
TRANSITION FROM schieben_work TO Blister_Out := #StateOk;
END_TRANSITION
STEP Blister_Out:
END_STEP
TRANSITION FROM Blister_Out TO Settling_Time := WTOut;
END_TRANSITION
STEP Settling_Time: (* min time T#2500ms; T#2500ms *)
END_STEP
TRANSITION FROM Settling_Time TO (Check_Verlaengerung_, check2) := TRUE;
END_TRANSITION
STEP Check_Verlaengerung_:
END_STEP
TRANSITION FROM Check_Verlaengerung_ TO VRZ_close := mit_Verlaengerung;
END_TRANSITION
TRANSITION FROM Check_Verlaengerung_ TO Step13 := TRUE;
END_TRANSITION
STEP VRZ_close:
	VRZ_close_action(N);
END_STEP
TRANSITION FROM VRZ_close TO Step13 := StateOk;
END_TRANSITION
STEP Step13:
END_STEP
STEP check2:
END_STEP
TRANSITION FROM check2 TO schieben_init := mit_schieben;
END_TRANSITION
TRANSITION FROM check2 TO Step14 := TRUE;
END_TRANSITION
STEP schieben_init:
	schieben_init_action(N);
END_STEP
TRANSITION FROM schieben_init TO Step14 := StateOk;
END_TRANSITION
STEP Step14:
END_STEP
TRANSITION FROM (Step13, Step14) TO SeqEnd := TRUE;
END_TRANSITION
STEP SeqEnd: (* -> WAIT *)
	SeqEnd_action(N);
END_STEP
TRANSITION FROM SeqEnd TO JumpAutoRun := TRUE;
END_TRANSITION

ACTION STATE_WAITFirstAutRun_action:
IF 		ModeSelect.Mode=MODE_AUTO_RUN
	OR 	ModeSelect.Mode=MODE_STEP_RUN
  OR SpecialMode01.State=State_Run
THEN
	State:=STATE_RUN;
	Result:=RESULT_NON;
ELSE
	State:=STATE_WAIT;
	SFCRun:=FALSE;
(*ELSE*)
END_IF
END_ACTION

ACTION STATE_WAITForAutoRun_entry:
Delay(In:=FALSE);
END_ACTION

ACTION STATE_WAITForAutoRun_action:
Delay(IN:=
	NOT ST08_400_B50_0.BitInToCheck AND
	ST08_401_B50_5.BitInToCheck AND
	ST08_400_Y50_2.InitPosition,
	PT:=T#1500ms);
IF 	((	ModeSelect.Mode=MODE_AUTO_RUN OR 	ModeSelect.Mode=MODE_STEP_RUN   OR SpecialMode01.State=State_Run  )
	AND Delay.Q )

THEN
	State:=STATE_RUN;
	Result:=RESULT_NON;
	SFCTimeStart:=TIME();
ELSE
	State:=STATE_WAIT;
END_IF
END_ACTION

ACTION VRZ_open_action:
ST08_400_Y50_0.MoveWork:=TRUE;
END_ACTION

ACTION schieben_work_action:
ST08_401_Y52_4.MoveWork:=TRUE;
END_ACTION

ACTION VRZ_close_action:
ST08_400_Y50_0.MoveInit:=TRUE;
END_ACTION

ACTION schieben_init_action:
ST08_401_Y52_4.MoveInit:=TRUE;
END_ACTION

ACTION SeqEnd_action:
SFCTime:=TIME_TO_DINT(TIME()-SFCTimeStart);
State:=STATE_WAIT;
END_ACTION

TRANSITION mit_Verlaengerung:
mp.ST08.Trayzufuhr_Verlaengerung
END_TRANSITION

TRANSITION StateOk:
ST08_400_Y50_0.State=STATE_OK
END_TRANSITION

TRANSITION mit_schieben:
MP.ST08.Traystapel_schieben AND
MP.ST08.Trayzufuhr_Verlaengerung
END_TRANSITION

TRANSITION #StateOk:
ST08_401_Y52_4.State=STATE_OK
END_TRANSITION

TRANSITION WTOut:
ST08_400_B50_0.BitInToCheck=TRUE AND ST08_401_B50_5.BitInToCheck=FALSE
END_TRANSITION

TRANSITION mit_Verlaengerung:
MP.ST08.Trayzufuhr_Verlaengerung
END_TRANSITION

TRANSITION StateOk:
ST08_400_Y50_0.State=STATE_OK
END_TRANSITION

TRANSITION mit_schieben:
MP.ST08.Traystapel_schieben AND
MP.ST08.Trayzufuhr_Verlaengerung
END_TRANSITION

TRANSITION StateOk:
ST08_401_Y52_4.State=STATE_OK
END_TRANSITION
END_PROGRAM

(* POU Stations/ST_08_Palettierer/ST_08_SFCs/Inlett/ST08_VV1_Y50_2, SFC *)
PROGRAM ST08_VV1_Y50_2				(* Vereinzler vor HQE4 *)

VAR_OUTPUT
	SFCCurrentPOU	: STRING:='ST08_VV1_Y50_2';
	SFCCurrentStep	: STRING:='';
	SFCTime			: DINT;
	State   		: DINT;
	Result  		: DINT;
END_VAR
VAR_INPUT

END_VAR
VAR
	MsgOK			: BOOL;
	MsgCancel		: BOOL;
	SFCRun			: BOOL;
	SFCTimeStart	: TIME;
	Delay			: TON;
	TimeOut			: TON;
	(* Userdefinded area *)

END_VAR
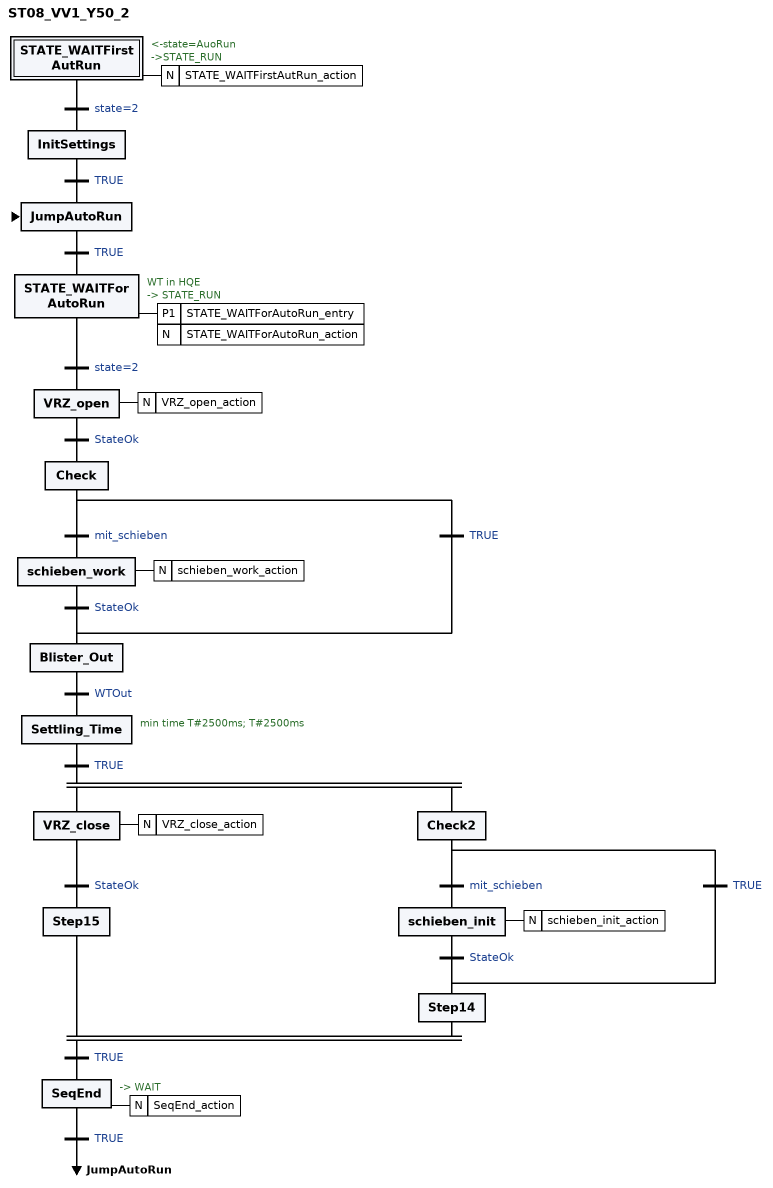
INITIAL_STEP STATE_WAITFirstAutRun: (* <-state=AuoRun / ->STATE_RUN *)
	STATE_WAITFirstAutRun_action(N);
END_STEP
TRANSITION FROM STATE_WAITFirstAutRun TO InitSettings := state=2;
END_TRANSITION
STEP InitSettings:
END_STEP
TRANSITION FROM InitSettings TO JumpAutoRun := TRUE;
END_TRANSITION
STEP JumpAutoRun:
END_STEP
TRANSITION FROM JumpAutoRun TO STATE_WAITForAutoRun := TRUE;
END_TRANSITION
STEP STATE_WAITForAutoRun: (* WT in HQE / -> STATE_RUN *)
	STATE_WAITForAutoRun_entry(P1);
	STATE_WAITForAutoRun_action(N);
END_STEP
TRANSITION FROM STATE_WAITForAutoRun TO VRZ_open := state=2;
END_TRANSITION
STEP VRZ_open:
	VRZ_open_action(N);
END_STEP
TRANSITION FROM VRZ_open TO Check := StateOk;
END_TRANSITION
STEP Check:
END_STEP
TRANSITION FROM Check TO schieben_work := mit_schieben;
END_TRANSITION
TRANSITION FROM Check TO Blister_Out := TRUE;
END_TRANSITION
STEP schieben_work:
	schieben_work_action(N);
END_STEP
TRANSITION FROM schieben_work TO Blister_Out := StateOk;
END_TRANSITION
STEP Blister_Out:
END_STEP
TRANSITION FROM Blister_Out TO Settling_Time := WTOut;
END_TRANSITION
STEP Settling_Time: (* min time T#2500ms; T#2500ms *)
END_STEP
TRANSITION FROM Settling_Time TO (VRZ_close, Check2) := TRUE;
END_TRANSITION
STEP VRZ_close:
	VRZ_close_action(N);
END_STEP
TRANSITION FROM VRZ_close TO Step15 := StateOk;
END_TRANSITION
STEP Step15:
END_STEP
STEP Check2:
END_STEP
TRANSITION FROM Check2 TO schieben_init := mit_schieben;
END_TRANSITION
TRANSITION FROM Check2 TO Step14 := TRUE;
END_TRANSITION
STEP schieben_init:
	schieben_init_action(N);
END_STEP
TRANSITION FROM schieben_init TO Step14 := StateOk;
END_TRANSITION
STEP Step14:
END_STEP
TRANSITION FROM (Step15, Step14) TO SeqEnd := TRUE;
END_TRANSITION
STEP SeqEnd: (* -> WAIT *)
	SeqEnd_action(N);
END_STEP
TRANSITION FROM SeqEnd TO JumpAutoRun := TRUE;
END_TRANSITION

ACTION STATE_WAITFirstAutRun_action:
IF 		ModeSelect.Mode=MODE_AUTO_RUN
	OR 	ModeSelect.Mode=MODE_STEP_RUN
  OR SpecialMode01.State=State_Run
THEN
	State:=STATE_RUN;
	Result:=RESULT_NON;
ELSE
	State:=STATE_WAIT;
	SFCRun:=FALSE;
(*ELSE*)
END_IF
END_ACTION

ACTION STATE_WAITForAutoRun_entry:
Delay(IN:=FALSE);
END_ACTION

ACTION STATE_WAITForAutoRun_action:
Delay(IN:=
	NOT ST08_401_B50_5.BitInToCheck AND
	ST08_402_B51_2.BitInToCheck AND
	ST08_402_Y50_4.InitPosition,
	PT:=T#1500ms);
IF 	((	ModeSelect.Mode=MODE_AUTO_RUN OR 	ModeSelect.Mode=MODE_STEP_RUN   OR SpecialMode01.State=State_Run  )
	AND Delay.Q )

THEN
	State:=STATE_RUN;
	Result:=RESULT_NON;
	SFCTimeStart:=TIME();
ELSE
	State:=STATE_WAIT;
END_IF
END_ACTION

ACTION VRZ_open_action:
ST08_400_Y50_2.MoveWork:=TRUE;
END_ACTION

ACTION schieben_work_action:
ST08_402_Y52_6.MoveWork:=TRUE;
END_ACTION

ACTION VRZ_close_action:
ST08_400_Y50_2.MoveInit:=TRUE;
END_ACTION

ACTION schieben_init_action:
ST08_402_Y52_6.MoveInit:=TRUE;
END_ACTION

ACTION SeqEnd_action:
SFCTime:=TIME_TO_DINT(TIME()-SFCTimeStart);
State:=STATE_WAIT;
END_ACTION

TRANSITION StateOk:
ST08_400_Y50_2.State=STATE_OK
END_TRANSITION

TRANSITION mit_schieben:
MP.ST08.Traystapel_schieben AND
MP.ST08.Trayzufuhr_Verlaengerung
END_TRANSITION

TRANSITION StateOk:
ST08_402_Y52_6.State=STATE_OK
END_TRANSITION

TRANSITION WTOut:
ST08_401_B50_5.BitInToCheck=TRUE AND ST08_402_B51_2.BitInToCheck=FALSE
END_TRANSITION

TRANSITION StateOk:
ST08_400_Y50_2.State=STATE_OK
END_TRANSITION

TRANSITION mit_schieben:
MP.ST08.Traystapel_schieben AND
MP.ST08.Trayzufuhr_Verlaengerung
END_TRANSITION

TRANSITION StateOk:
ST08_402_Y52_6.State=STATE_OK
END_TRANSITION
END_PROGRAM

(* POU Stations/ST_00/ST00_PRGs/_CallPRGs, ST *)
PROGRAM _CallPRGs
VAR
END_VAR
ST00_CallPRGs();
ST02_CallPRGs();
ST03_CallPRGs();
ST08_CallPRGs();
END_PROGRAM

(* POU Stations/ST_00/ST00_PRGs/ST00_CallPRGs, ST *)
PROGRAM ST00_CallPRGs
VAR
	FB_ReadXmlLineConf		: FB_ReadXmlLine;
	sDescription			: STRING;
END_VAR
Lights_and_Lamps();
Safety_Fuses_AirPressure();
JobManagement();
VisuLogger();

IF 	HomePositionSFC.State = STATE_RUN THEN
	ListHomeNOK(InstName:='ST00 ',Description:=sDescription);
END_IF
FB_ReadXmlLineConf(
	Prefix:= 'CONFIG',
	ID:= 'ST00',
	File:= 'CONFIG.xml',
	Text=> sDescription );


IF gInitOk AND ST_Path.Done THEN
	MachineStates();
	ST_Service();
	ST00_ImpExp_MP(
				path:= MP_LocalDriveRoot,
				filename	:=MP_MPExportFilename);
END_IF

(* Schutztüren *)
IF 	ModeSelect.Mode>MODE_MANUAL AND
	ST00_220_S1.BitInToCheck THEN
	ModeSelect.AskForManual:=TRUE;

END_IF

IF	ModeSelect.Mode>MODE_MANUAL THEN
	ST00_220_S1_S31.SetSignalHigh:=TRUE;
	ST00_245_V1.SetSignalHigh:=TRUE;
END_IF

IF 	ModeSelect.Mode<=MODE_MANUAL THEN
	ST00_220_S1_S31.SetSignalLow:=TRUE;
	ST00_245_V1.SetSignalLow:=TRUE;
END_IF

(* Generierung RoboterOffset *)
gRobotOffset :=  TD.RobotOffset;

gTypeCode:=STRING_TO_DINT(DELETE(TD.TypeCode,1,1));
END_PROGRAM

(* POU Stations/ST_00/ST00_PRGs/Lights_and_Lamps, ST *)
PROGRAM Lights_and_Lamps
VAR
	SignalRed			: BOOL;
	SignalOrange		: BOOL;
	SignalGreen			: BOOL;
	SignalBlue			: BOOL;
	SetOrange			: BOOL;
	FP_MachineLight	: R_TRIG;
	FN_MachineLight	: F_TRIG;
	PartLack			: TON;
	TimeOFF			: TON;
	fb_Blinker			: FB_Blinker;
END_VAR
fb_Blinker(b_start:=TRUE, t_taktzeit_on:=t#1s , t_taktzeit_off:=t#1s , b_blinker_out=> );
(* ----------------------------------------------------------------------------------------- *)
(* Ampel  *)
SignalRed	:= ErrorHandler.bOutError ;
SignalOrange	:= MessageHandler.MessageActive OR SetOrange OR ST03_Test_Parts.fb_Blinker.b_blinker_out;;
IF	ModeSelect.Mode=MODE_AUTO_RUN OR ModeSelect.Mode=MODE_STEP_RUN THEN
	SignalGreen	:=TRUE;
ELSIF
	 ModeSelect.Mode=MODE_AUTO_STOP THEN
	SignalGreen	:=fb_Blinker.b_blinker_out;
ELSE
	SignalGreen	:=FALSE;
END_IF
(*SignalGreen	:= ModeSelect.Mode=MODE_AUTO_RUN OR ModeSelect.Mode=MODE_AUTO_STOP OR ModeSelect.Mode=MODE_STEP_RUN;*)
SignalBlue	:= FALSE; (* Parts Missing *)

(* ----------------------------------------------------------------------------------------- *)
PartLack(IN:= FALSE,PT:=T#60s);
IF  	ModeSelect.Mode>MODE_MANUAL AND
	PartLack.Q THEN
	SetOrange:=TRUE;
ELSE
	SetOrange:=FALSE;
END_IF

IF	CurrentVisu <> 'MANUAL_ST00_0' THEN

	(* Ampel Grün *)
	IF 	ST00_350_H1.State=STATE_WAIT AND
		ST00_350_H1.SignalOut <> SignalRed THEN
		ST00_350_H1.SetSignalHigh:= SignalRed;
		ST00_350_H1.SetSignalLow:= NOT SignalRed;
	END_IF;

	(* Ampel Orange *)
	IF 	ST00_350_H2.State=STATE_WAIT AND
		ST00_350_H2.SignalOut <> SignalOrange	THEN
		ST00_350_H2.SetSignalHigh:= SignalOrange;
		ST00_350_H2.SetSignalLow:= NOT SignalOrange;
	END_IF;
	(* Ampel Rot *)
	IF 	ST00_350_H3.State=STATE_WAIT AND
		ST00_350_H3.SignalOut <> SignalGreen THEN
		ST00_350_H3.SetSignalHigh:= SignalGreen;
		ST00_350_H3.SetSignalLow:= NOT SignalGreen;
	END_IF;
	(*Ampel Blau*)
	(*IF 	ST00_350_H4.State=STATE_WAIT AND
		ST00_350_H4.SignalOut <> SignalBlue THEN
		ST00_350_H4.SetSignalHigh:= SignalBlue;
		ST00_350_H4.SetSignalLow:= NOT SignalBlue;
	END_IF*)

(* Bedientaster-Beleuchtungen *)
	(* H3 Reset *)
	IF 	ST00_292_H3_RESET.State=STATE_WAIT AND
		ST00_292_H3_RESET.SignalOut <> SignalRed THEN
		ST00_292_H3_RESET.SetSignalHigh:=SignalRed;
		ST00_292_H3_RESET.SetSignalLow:= NOT SignalRed;
	END_IF;
	(* H2 Start *)
	IF 	ST00_292_H2_Start.State=STATE_WAIT AND
		ST00_292_H2_Start.SignalOut <> SignalGreen 	THEN
		ST00_292_H2_Start.SetSignalHigh:=SignalGreen;
		ST00_292_H2_Start.SetSignalLow:= NOT SignalGreen;
	END_IF

	(* H3 Reset *)
	IF 	ST00_245_V3_RESET.State=STATE_WAIT AND
		ST00_245_V3_RESET.SignalOut <> SignalRed THEN
		ST00_245_V3_RESET.SetSignalHigh:=SignalRed;
		ST00_245_V3_RESET.SetSignalLow:= NOT SignalRed;
	END_IF;
	(* H2 Start *)
	IF 	ST00_245_V2_START.State=STATE_WAIT AND
		ST00_245_V2_START.SignalOut <> SignalGreen 	THEN
		ST00_245_V2_START.SetSignalHigh:=SignalGreen;
		ST00_245_V2_START.SetSignalLow:= NOT SignalGreen;
	END_IF
END_IF

(* Beleuchtung Anlage Ein, wenn Schutz geöffnet*)
(* ----------------------------------------------------------------------------------------- *)

(* Flag Positive - Light on*)
FP_MachineLight(CLK:=NOT gReadyForControlOn );

(* Flag Negative - Light on*)
FN_MachineLight(CLK:=NOT gReadyForControlOn );

TimeOFF(IN:=ST00_31_K1.SignalOut, PT:=t#5m);

IF 	FP_MachineLight.Q THEN
	ST00_31_K1.SetSignalHigh	:= TRUE;
	ST00_31_K1.SetSignalLow	:= FALSE;
END_IF
IF 	FN_MachineLight.Q OR
	TimeOFF.Q THEN
	ST00_31_K1.SetSignalHigh	:= FALSE;
	ST00_31_K1.SetSignalLow	:= TRUE;
END_IF
END_PROGRAM

(* POU zLibrary/ept/Funktionsbausteine/FB_Blinker, ST *)
FUNCTION_BLOCK FB_Blinker
VAR_INPUT
	b_start 		: BOOL;
	t_taktzeit_on	: TIME;
	t_taktzeit_off	: TIME;
END_VAR
VAR_OUTPUT
	b_blinker_out : BOOL;
END_VAR
VAR
	fb_ton		: TON;
END_VAR
fb_ton(IN:=NOT fb_ton.Q AND b_start , PT:=t_taktzeit_off + t_taktzeit_on , Q=> , ET=> );
b_blinker_out:= fb_ton.ET >= t_taktzeit_off;
END_FUNCTION_BLOCK

(* POU Stations/ST_03_Ruestsaetze/ST_03_SFCs/ST03_Test_Parts, ST *)
PROGRAM ST03_Test_Parts
VAR
	FB_Blinker					: FB_Blinker;
END_VAR
(* An der Oberfläche muss bestätigt werden, dass die Prüfteile entnommen worden sind *)
IF 	gTakeTestPartsFinished OR
	ST_CPU.LNG <> CZ THEN
	ST03_Main.TestPartsRemove := FALSE;
END_IF

(* Meldung blinken bis Teile entnommen werden / Blikani okna odeber vzorky do potvrzeni odebrani*)
fb_Blinker(b_start:=ST03_Main.TestPartsRemove , t_taktzeit_on:=t#1s , t_taktzeit_off:=t#1s , b_blinker_out=> );

(*Beim Dummytest 160 polig dürfen die Isos nicht bedruckt werden
	/ Stop Printing at Dummytest 160 pol*)

IF	gTypeCode=322	THEN 	(*160 polig*)
	IF 	NOT DummyTest_160pol THEN
		IF	ST03_8_B76_1.BitInToCheck OR  (* 3621 *)
			ST03_423_B66_0.BitInToCheck THEN (* Rüstsatz 160 polig LS 1 *)
			ST03_PLAN_70V1_1.SetSignalHigh	:= TRUE;		(* Start  Bedrucken Tintenstrahldrucker Frontseite*)
			ST03_PLAN_70V1_1.SetSignalLow	:= FALSE;
		ELSE
			ST03_PLAN_70V1_1.SetSignalHigh	:= FALSE;	(* Start  Bedrucken Tintenstrahldrucker Frontseite*)
			ST03_PLAN_70V1_1.SetSignalLow	:= TRUE;
		END_IF
		IF	ST03_8_B76_2.BitInToCheck OR (* 3621 *)
			ST03_422_B64_0.BitInToCheck THEN  (* Rüstsatz 160 polig LS 2 *)
			ST03_PLAN_71V1_2.SetSignalHigh	:= TRUE;		(* Start  Bedrucken Tintenstrahldrucker Rückseite*)
			ST03_PLAN_71V1_2.SetSignalLow	:= FALSE;
		ELSE
			ST03_PLAN_71V1_2.SetSignalHigh	:= FALSE;	(* Start  Bedrucken Tintenstrahldrucker Rückseite*)
			ST03_PLAN_71V1_2.SetSignalLow	:= TRUE;
		END_IF
	END_IF
END_IF

	(*  Nur in CZ
	Bei erreichen der vorgegebenen Stückzahl werden automatisch Testteile abgelegt
	Spusteni vzorku pri dosazeni zadane hodnoty *)

IF 	ST_CPU.LNG = CZ AND
	NOT MP.ST02.DummyPruefung_93pol THEN
	IF 	gPartsTest >= gPartsTestVisu AND
		NOT gTakeTestPartsAuto	THEN
		gTakeTestPartsAuto:=TRUE;
	END_IF

	IF 	gPartsTest >= gPartsTestVisu THEN
		gPartsTest:=0;
	END_IF
ELSE
	gTakeTestPartsAuto:=FALSE;
	IF 	gTakeTestParts  THEN
		gPartsTest:=0;
	END_IF
END_IF
END_PROGRAM

(* POU Stations/ST_00/ST00_PRGs/JobManagement, ST *)
PROGRAM JobManagement
VAR
	(*Buttons*)
	BtnOffsetPlus				: VisuButton;
	VisuBtnOffsetPlus			: sButtonVisu;
	BtnOffsetMinus				: VisuButton;
	VisuBtnOffsetMinus			: sButtonVisu;
	BtnClearAll					: VisuButton;
	VisuBtnClearAll				: sButtonVisu;
	BtnTestParts				: VisuButton;
	VisuBtnTestParts			: sButtonVisu;

END_VAR
(*Gesamt-IO zuweisen, Gesamt-NIO ermitteln
  ---------------------------------------------------------------------------------*)
MP.ST00.PartsNokTotal:=0;
(*
FOR StIdx:=1 TO NO_OF_NEST
DO
	MP.ST00.PartsNokTotal:=MP.ST00.PartsNokTotal+MP.ST00.PartsNok_ST02[StIdx];
END_FOR
*)
MP.ST00.PartsNokTotal:=0;
MP.ST00.PartsOkTotal:=0;

(*Noch zu produzierende Teile ermitteln
  ---------------------------------------------------------------------------------*)
MP.ST00.PartsRemaining:=(		MP.ST00.PartsToProduce
										 		+ 	MP.ST00.PartsToProduceOffset
										 		- 	gPartsInserted
										 													);

(*Korrekturwert für Sollstückzahl erhöhen bzw verringern
  ---------------------------------------------------------------------------------*)
BtnOffsetPlus(Button:=VisuBtnOffsetPlus,
							Enable:=TRUE,
							Visible:=TRUE,
							TextOn:='+',
							);
BtnOffsetMinus(	Button:=VisuBtnOffsetMinus,
								Enable:=MP.ST00.PartsToProduceOffset>0,
								Visible:=TRUE,
								TextOn:='-');

IF BtnOffsetPlus.PressedFlag THEN
	MP.ST00.PartsToProduceOffset:=MP.ST00.PartsToProduceOffset+1;
END_IF
IF BtnOffsetMinus.PressedFlag THEN
	MP.ST00.PartsToProduceOffset:=MP.ST00.PartsToProduceOffset-1;
END_IF

(*Alle Zähler löschen
  ---------------------------------------------------------------------------------*)
BtnClearAll(Button:=VisuBtnClearAll,
						Enable:=TRUE,
						Visible:=TRUE,
						TextOn:='Alle Zähler löschen',
						);
IF BtnClearAll.PressedFlag THEN
	MP.ST00.PartsToProduce:=0;
	MP.ST00.PartsToProduceOffset:=0;
	MP.ST00.PartsNokSubsetSize:=0;
	gPartsInserted:=0;
	gNokPartsColorCam:=0;
	gNokPartsWingCam:=0;
	gNokPartsPrint:=0;
	NokCounter1li:= 0;
	NokCounter1re:= 0;
	NokCounter2li:= 0;
	NokCounter2re:= 0;
	NokCounter3li:= 0;
	NokCounter3re:= 0;
	i32_first_parts :=0;
END_IF

(*Test Teile entnehmen
  ---------------------------------------------------------------------------------*)
BtnTestParts(	Button:=VisuBtnTestParts,
						Enable:=TRUE,
						Visible:=ModeSelect.Mode=MODE_AUTO_RUN AND
								NOT ST03_Main.TestPartsRemove,
						TextOn:='TestParts',
				);

IF 	ModeSelect.Mode=MODE_AUTO_RUN AND BtnTestParts.PressedFlag THEN
  	gTakeTestParts:=TRUE;
ELSIF
	ModeSelect.Mode<>MODE_AUTO_RUN THEN
	gTakeTestParts:=FALSE;
END_IF
END_PROGRAM

(* POU Stations/ST_00/ST00_PRGs/VisuLogger, ST *)
PROGRAM VisuLogger
VAR
	PageHistory		: ARRAY[1..20] OF STRING(40);
	Trigger				: BOOL;
	Clock					: R_TRIG;
	LastVisuPage	: STRING(40);
	bDeleteBuf		: BOOL;
	i							: INT;
END_VAR
IF 	LastVisuPage='' THEN
	LastVisuPage:=CurrentVisu;
END_IF

Trigger:=CurrentVisu<>LastVisuPage;
Clock(Clk:=Trigger);

IF 	Clock.Q THEN
	FOR i:= 20 TO 2 BY -1 DO
		PageHistory[i]:=PageHistory[i-1];
	END_FOR
	PageHistory[1]:=CurrentVisu;
END_IF

IF 	bDeleteBuf THEN
	FW_MemSet(ADR(PageHistory), 0, SIZEOF(PageHistory));
	bDeleteBuf:=FALSE;
END_IF

LastVisuPage:=CurrentVisu;
END_PROGRAM

(* POU Stations/ST_00/ST00_PRGs/MachineStates, ST *)
PROGRAM MachineStates
VAR
	InfoNoUser				: ErrorStruct;
	LogFileEntry			: ErrorStruct;
	FP_AutoRun				: R_TRIG;
	FirstCycle				: BOOL := TRUE;
	FP_STOP					: R_TRIG;
	TON_STOP				: TON;
	CycleTime             	: REAL;
	CycleTimeHelp           : STRING;

	FB_ReadXmlLineMsg		: FB_ReadXmlLine;
	FB_ReadXmlLineUser		: FB_ReadXmlLine;

	s_MsgNew				: STRING;
	s_UserNew				: STRING;
END_VAR
(* Programmaufrufe *)
_Message();

(*Open Main-Screen with AutoStart-Button*)
FP_AutoRun(CLK:= ModeSelect.Mode=MODE_AUTO);

IF FP_AutoRun.Q THEN
	CurrentVisu:='MAIN';
END_IF

(* SYSTEM_GST *)
IF ModeSelect.HomePosRunFirstImp THEN
	CurrentVisu:='SYSTEM_GST';
END_IF


(*Button "Leerfahren" einblenden*)
ModeSelect.ShowBtnRunEmpty:=TRUE;

(*Taster "Start" und "Stop" am Schaltschrank*)
IF 	(ModeSelect.Mode<=MODE_MANUAL AND ModeSelect.BtnManual.Visible OR ModeSelect.Mode=MODE_AUTO)AND
	(ST00_292_S2_START.BitInToCheck OR ST00_245_S2_START.BitInToCheck) THEN
	ModeSelect.iRemoteAutoStart:=TRUE;
END_IF

FP_STOP(CLK:=ST00_292_S1_STOP.BitInToCheck OR ST00_245_S1_STOP.BitInToCheck);

IF 	ModeSelect.Mode=MODE_AUTO_RUN AND
	FP_STOP.Q THEN
	ModeSelect.iRemoteAutoStop:=TRUE;
END_IF

IF 	ModeSelect.Mode=MODE_AUTO AND
	FP_STOP.Q THEN
	ModeSelect.AskForManual:=TRUE;
END_IF


CycleTime:=DINT_TO_REAL (ST03_Main.SFCTime);

CycleTime:=(CycleTime/10000);
CycleTimeHelp:=REAL_TO_STRING(CycleTime);
CycleTimeHelp:=LEFT(CycleTimeHelp,4);

(* Force ManualMode if AutoStop not successful *)
TON_STOP(IN:=ST00_292_S1_STOP.SignalIn OR ST00_245_S1_STOP.SignalIn, PT:=t#1s );
IF 	ModeSelect.Mode=MODE_AUTO_STOP AND
	TON_STOP.Q THEN
	ModeSelect.AskForManual:=TRUE;
END_IF

(*Force HomePosition-Run after every Manual-Mode*)
IF 	ModeSelect.Mode<=MODE_MANUAL THEN
	gHomePosSFCDone:=FALSE;
END_IF

IF 	ModeSelect.Mode<>MODE_Special THEN
	DummyTest_160pol := FALSE;
	MP.ST02.DummyPruefung_93pol :=FALSE;
END_IF
END_PROGRAM
ACTION _Message:
(* setze Dateinamen für Fehlerdatei *)
ErrorHandler.ErrorLogFileName := CONCAT(LOG_RDPathLocal,'ErrorLog_');
ErrorHandler.ErrorLogFileName := CONCAT(ErrorHandler.ErrorLogFileName, WORD_TO_STRING(CallGeneralFunctions.wYear));
ErrorHandler.ErrorLogFileName := CONCAT(ErrorHandler.ErrorLogFileName, '-');
ErrorHandler.ErrorLogFileName := CONCAT(ErrorHandler.ErrorLogFileName, WORD_TO_STRING(CallGeneralFunctions.wMonth));
ErrorHandler.ErrorLogFileName := CONCAT(ErrorHandler.ErrorLogFileName, '.csv');



(*LogFile-Eintrag bei Betriebsarten-Umschaltung*)
IF 	FirstCycle THEN
	FB_ReadXmlLineMsg.ID:='bm_restart';
	FirstCycle:=FALSE;
ELSIF
	ModeSelect.ManualFirstImp THEN
	FB_ReadXmlLineMsg.ID:='bm_manual_mode';
ELSIF
	ModeSelect.AutoFirstImp THEN
	FB_ReadXmlLineMsg.ID:='bm_automatic_mode';
ELSIF
	ModeSelect.HomePosRunFirstImp THEN
	FB_ReadXmlLineMsg.ID:='bm_homepos';
END_IF

IF	s_MsgNew <> FB_ReadXmlLineMsg.Text AND
	FB_ReadXmlLineMsg.Text <> '' THEN
	LogFileEntry.DateTime:=gVarDTSystemtime;
	LogFileEntry.Text  	:=FB_ReadXmlLineMsg.Text;
	LogFileEntry.Typ   	:=1; (*yellow Info-Line*)
	LogFileEntry.No    	:=1;
	ErrorHandler.AddError(ErrorToAdd:=LogFileEntry,sVisu:=Visu.ErrorHandler);
	s_MsgNew:=FB_ReadXmlLineMsg.Text;
END_IF



(*Show a Message when no User is logged in*)
IF	NOT UserLoginHandler.UserLoggedIn THEN
	FB_ReadXmlLineUser.ID:='bm_user_not_login';
END_IF

IF	s_UserNew <> FB_ReadXmlLineUser.Text AND
	FB_ReadXmlLineUser.Text <> '' THEN
	InfoNoUser.DateTime:=gVarDTSystemtime;
	InfoNoUser.Text  	:=FB_ReadXmlLineUser.Text;
	InfoNoUser.Typ   	:=2; (*yellow Info-Line*)
	InfoNoUser.No    	:=1;
	ErrorHandler.AddError(ErrorToAdd:=InfoNoUser,sVisu:=Visu.ErrorHandler);
	s_UserNew:=FB_ReadXmlLineUser.Text;
END_IF



(*Aufrufe*)
FB_ReadXmlLineMsg(
	Prefix:= 'MSG',
	File:= 'MSG.xml');

FB_ReadXmlLineUser(
	Prefix:= 'MSG',
	File:= 'MSG.xml');
END_ACTION

(* POU zLibrary/ept/Service/ST_Service, ST *)
PROGRAM ST_Service
VAR_INPUT
	st_ctrl_in						: struct_ctrl_in;
END_VAR
VAR_OUTPUT
	Error							:BOOL;
	ErrorMsg: STRING(255);	(*  *)
	ErrorID					:STRING(20);
END_VAR
VAR
	b_first_cycle					: BOOL := TRUE;
	fb_state_entry				: ST_StateEntry;

	fb_ton_uez						: TON;
	fb_ton_wz									: TON;
	fb_r_trig_counter					:R_TRIG;
	i_aktueller_tag						: INT;
	lr_aktuelle_stunden				: LREAL;
	i_aktuelle_stunden				: INT;
	MsgOK											:BOOL;
	fb_bbgen_xml_file					: ST_BBGenXMLFile;
	Service_daten_copy				: ARRAY [0..15] OF struct_daten_service;
	betriebssekundenzaehler_copy	:UDINT;
	M_BtnType									: ARRAY[0..15] OF BOOL;
	HelpString						:STRING(255);
	FB_Betriebsstundenzaehler	:FB_Betriebsstundenzaehler;
	lr_Betriebsstunden					:LREAL;
	Start								:BOOL;
	gPartsInsertedCopy				: DINT;
	i_act_ErrorNumber				:INT;
	ColorName							: ARRAY[0..15] OF DINT; (*from STRUCT Colors*)
	Default_reached						: ARRAY[0..15] OF BOOL; 	 (*Merker damit Fehlermeldung nur einmal angezeigt wird*)
	Warning_reached						: ARRAY[0..15] OF BOOL;	(*Merker damit Warnmeldung nur einmal angezeigt wird*)
	Reset_Help						: ARRAY[1..3] OF BOOL;

	CURRENTLANGUAGECopy			: STRING(5);

	fb_ExpActService				: FB_ExporString;	(* Fehlermeldungen in Errorlog (txt) schreiben *)
END_VAR
VAR_TEMP
	i					:INT:=-1;
	k					:INT:=-1;
END_VAR
Reset();

FB_Betriebsstundenzaehler(
	Start:= ModeSelect.Mode=MODE_AUTO_RUN OR Start,
	Reset:= ,
	i32_betriebssekundenzaehler_in:= Service.betriebssekundenzaehler,
	i32_betriebssekundenzaehler=> Service.betriebssekundenzaehler,
	lr_betriebsstundenzaehler=> lr_Betriebsstunden);

(*Zeiten*)
fb_ton_uez(IN:= , PT:= , Q=> , ET=> );
fb_ton_wz(IN:= , PT:= , Q=> , ET=> );

(*Flanken*)
fb_r_trig_counter(CLK:= gPartsInsertedCopy<>gPartsInserted, Q=> );	(*ST02_160_A1_3.BitOutToSet	 Signal von Rundschalttisch drehen *)
gPartsInsertedCopy:=gPartsInserted;

(* Hochzählen der einelnen Zähler *)
IF fb_r_trig_counter.Q THEN
	FOR i:=0 TO 15 BY 1 DO
		IF Service.daten[i].Type_Service = COUNTER AND Service.daten[i].Default_Value > 0 THEN
			Service.daten[i].Current_Value := Service.daten[i].Current_Value +1;
		END_IF
	END_FOR
END_IF

(* Tage seit dem 01.01.2000 *)
i_aktueller_tag := (WORD_TO_INT (gVarSystemtime.wYear) - 2000) *360;	(* Anzahl der Jahre x360 Tage *)
i_aktueller_tag := i_aktueller_tag + (WORD_TO_INT (gVarSystemtime.wMonth)*30) ;	(* Anzahl der Monate x30 Tage *)
i_aktueller_tag := i_aktueller_tag + WORD_TO_INT (gVarSystemtime.wDay);	(* Anzahl der Tage *)

lr_aktuelle_stunden:=WORD_TO_LREAL(gVarSystemtime.wHour)+
										(WORD_TO_LREAL(gVarSystemtime.wMinute)/60);		(*Anzahl der Stunden*)
i_aktuelle_stunden:=LREAL_TO_INT(lr_aktuelle_stunden*100);
lr_aktuelle_stunden:=INT_TO_LREAL(i_aktuelle_stunden)/100;


Umschalten();

(*===================================================================================================================================*)

(* Toplevel *)
IF fb_state_entry.i16_next_step > INIT AND fb_state_entry.i16_next_step < FEHLER THEN
	IF fb_state_entry.i16_next_step < STOP THEN
		IF st_ctrl_in.b_stop THEN
			fb_state_entry.i16_next_step := STOP;
		END_IF
	END_IF
END_IF


fb_state_entry(i16_pos:= 1);

CASE fb_state_entry.i16_step OF
(*=======================================================*)
	INIT_OBJ:

		IF 	b_first_cycle THEN	(* Programmstart >> XML Datei auslesen *)
			fb_state_entry.i16_next_step := 200;
		ELSE
			fb_state_entry.i16_next_step := INIT;
		END_IF

(*=======================================================*)
	INIT:
		IF fb_state_entry.E THEN
			i := -1;
			Error := FALSE;
			fb_bbgen_xml_file.start_lesen_service := FALSE;
			fb_bbgen_xml_file.start_schreiben_service := FALSE;
			FOR i:=0 TO 15 BY 1 DO
				ColorName[i]:=color.white;
				Service.daten[i].Warning_reached := FALSE;
				Service.daten[i].Default_reached := FALSE;
			END_FOR
		END_IF

		(*-----------------------Weiterschaltbedingungen----------------------------*)
		IF NOT fb_state_entry.E THEN
			fb_state_entry.i16_next_step := BEREIT;
		END_IF

(*=======================================================*)
	BEREIT:		fb_state_entry.s_debugtext:='warte auf Änderung oder Sprachumschaltung';

		IF 	fb_state_entry.E AND i_act_ErrorNumber<> -1THEN
			ColorName[i_act_ErrorNumber]:=color.white;
			i_act_ErrorNumber:=-1;
		END_IF

		(*-----------------------Weiterschaltbedingungen----------------------------*)
		i := -1;
		FOR i:=0 TO 15 BY 1 DO

		(* Wenn Vorgabewert erreicht wird und der Start Button betätigt wird, wird eine Meldung ausgegeben *)
			IF 	Service.daten[i].Default_reached AND
				i_act_ErrorNumber =-1 AND
				NOT Default_reached[i]  THEN

					ErrorMsg:= CONCAT (Service.daten[i].Name, ' Vorgabewert erreicht');
					Default_reached[i]:=TRUE;
					i_act_ErrorNumber:=i;
					ColorName[i]:=color.lightgrey;
					fb_state_entry.i16_next_step:=FEHLER;

			END_IF

		(* Wenn Warngrenze erreicht wird und der Start Button betätigt wird, wird eine Meldung ausgegeben *)
			IF 	Service.daten[i].Warning_reached  AND
				i_act_ErrorNumber =-1 AND
				NOT Service.daten[i].Default_reached AND
				NOT Warning_reached[i] THEN

					Warning_reached[i]:=TRUE;
					i_act_ErrorNumber:=i;
					ErrorID:='';
					ErrorMsg:= CONCAT (Service.daten[i].Name, ' Warngrenze erreicht');
					ColorName[i]:=color.lightgrey;
					fb_state_entry.i16_next_step:=STOP;

			END_IF
		END_FOR

		IF	CURRENTLANGUAGECopy <> CURRENTLANGUAGE THEN
			fb_state_entry.i16_next_step := 200;
		END_IF

		(* Wenn Unterschied und im Handbetrieb, dann schreibe XML *)
		IF 	(MEMCMP(ADR(Service_daten_copy), ADR(Service.daten), SIZEOF(Service_daten_copy)) <> 0 ) AND
			(ModeSelect.Mode = MODE_MANUAL OR ModeSelect.Mode = MODE_NON) OR
			betriebssekundenzaehler_copy <> service.betriebssekundenzaehler THEN
			fb_bbgen_xml_file.start_lesen_service := FALSE;
			fb_bbgen_xml_file.start_schreiben_service := FALSE;
			fb_state_entry.i16_next_step:=110;
		END_IF

(*=======================================================*)
	110:	fb_state_entry.s_debugtext:='XML Schreiben';

		IF fb_state_entry.E THEN
			fb_bbgen_xml_file.start_schreiben_service := TRUE;
			fb_bbgen_xml_file.s_path := MP_TDPathService;
			fb_bbgen_xml_file.s_service := CONCAT(CURRENTLANGUAGE,'_Service');
		END_IF

		(*-----------------------Weiterschaltbedingungen----------------------------*)
		IF fb_bbgen_xml_file.fertig_schreiben AND NOT fb_state_entry.E THEN
			fb_bbgen_xml_file.start_schreiben_service := FALSE;
			Service_daten_copy := Service.daten;
			betriebssekundenzaehler_copy:=service.betriebssekundenzaehler;
			fb_state_entry.i16_next_step := BEREIT;
		ELSIF fb_bbgen_xml_file.bError THEN
			ErrorID:='PM1';
			ErrorMsg:= ' Fehler beim Schreiben der Service XML-Datei';
			fb_state_entry.i16_next_step := FEHLER;
		END_IF

(*=======================================================*)
	200:	fb_state_entry.s_debugtext:=CONCAT(CURRENTLANGUAGE,'_Servie.xml einlesen');

		IF fb_state_entry.E THEN
			fb_bbgen_xml_file.start_lesen_service := TRUE;
			fb_bbgen_xml_file.s_path := MP_TDPathService;
			fb_bbgen_xml_file.s_service := CONCAT(CURRENTLANGUAGE,'_Service');
			fb_ExpActService.Start:=TRUE;
		END_IF

		(*-----------------------Weiterschaltbedingungen----------------------------*)
		IF fb_bbgen_xml_file.fertig_lesen AND NOT fb_state_entry.E THEN
			CURRENTLANGUAGECopy:=CURRENTLANGUAGE;
			fb_bbgen_xml_file.start_lesen_service := FALSE;
			Service_daten_copy := Service.daten;
			betriebssekundenzaehler_copy:=service.betriebssekundenzaehler;
			Button_Init();
			b_first_cycle := FALSE;
			fb_state_entry.i16_next_step := INIT;
		ELSIF
			fb_bbgen_xml_file.bError OR fb_bbgen_xml_file.nErrId  <> 0 THEN
			ErrorID:='PM2';
			ErrorMsg:= '';
			ErrorMsg:= ' Fehler beim Lesen der Service XML-Datei';
			fb_state_entry.i16_next_step := FEHLER;
		END_IF

(*=======================================================*)
	FEHLER:
		IF fb_state_entry.E THEN
			MessageHandler.ClearMessageLines(sVisu:=Visu.Message);
		END_IF
		MessageHandler.Msg.ID:=ErrorID;
		MessageHandler.Msg.Color:=Color.red;
		MessageHandler.Msg.Name:='Service Error';
		MessageHandler.Msg.Text:=CONCAT(MessageHandler.Msg.Text,ErrorMsg);
		MessageHandler.Msg.Station:=0;

		MessageHandler(
			Prio:=2, 							(*1=highest, .. , 4=lowest*)
			Btn1Addr:=ADR(MsgOk),	(*Address of Button1 , if Zero then Button is unvisible*)
			Btn2Addr:=,						(*Address of Button2 , if Zero then Button is unvisible*)
			sVisu:=Visu.Message);
			(*-----------------------Weiterschaltbedingungen----------------------------*)
		IF MsgOK THEN
				MsgOk:=FALSE;
				ErrorMsg:='';
				fb_state_entry.i16_next_step:=0;
		END_IF

		Error := TRUE;

(*=======================================================*)
	STOP:
		IF fb_state_entry.E THEN
			MessageHandler.ClearMessageLines(sVisu:=Visu.Message);
		END_IF
		(* WARNUNG *)
		MessageHandler.Msg.ID:=ErrorID;
		MessageHandler.Msg.Color:=Color.yellow;
		MessageHandler.Msg.Name:='Service Warnung';
		MessageHandler.Msg.Text:=CONCAT(MessageHandler.Msg.Text,ErrorMsg);
		MessageHandler.Msg.Station:=0;


		MessageHandler(
			Prio:=2, 							(*1=highest, .. , 4=lowest*)
			Btn1Addr:=ADR(MsgOk),	(*Address of Button1 , if Zero then Button is unvisible*)
			Btn2Addr:=,						(*Address of Button2 , if Zero then Button is unvisible*)
			sVisu:=Visu.Message);
			(*-----------------------Weiterschaltbedingungen----------------------------*)
		IF MsgOK THEN
				MsgOk:=FALSE;
				ErrorMsg:='';
				fb_state_entry.i16_next_step:=0;
		END_IF

END_CASE

fb_state_entry(i16_pos:= 2);

fb_bbgen_xml_file(
	start_lesen_service:= ,
	start_schreiben_service:= ,
	s_path:= ,
	s_service:= ,
	fertig_lesen=> ,
	fertig_schreiben=> ,
	bError=> ,
	nErrId=> );


fb_ExpActService(
	Start:= ,
	ExportStr:=CONCAT(CURRENTLANGUAGE,'_Service.xml') ,
	FileName:= 'ActService.txt',
	Path:=  s_tools_path,
	Mode:=FOPEN_MODEWRITE,
	Busy=> ,
	Done=> ,
	Error=> ,
	ErrorMsg=> );
END_PROGRAM
ACTION Button_Init:
(*=====================================================================*)
FOR i:=0 TO 15 BY 1 DO
	Service.visu[i].BtnReset.Text := 'Reset';
	Service.visu[i].BtnReset.Enable := TRUE;
	Service.visu[i].BtnReset.BackgroundColor := Color.lightgrey;
	Service.visu[i].BtnReset.TextColor := Color.black;
	Service.visu[i].BtnReset.Visible := TRUE;


(*=====================================================================*)

	Service.visu[i].BtnStart.Text := 'Start';
	Service.visu[i].BtnStart.Enable := TRUE;
	Service.visu[i].BtnStart.BackgroundColor := Color.lightgrey;
	Service.visu[i].BtnStart.TextColor := Color.black;
	Service.visu[i].BtnStart.Visible := TRUE;


